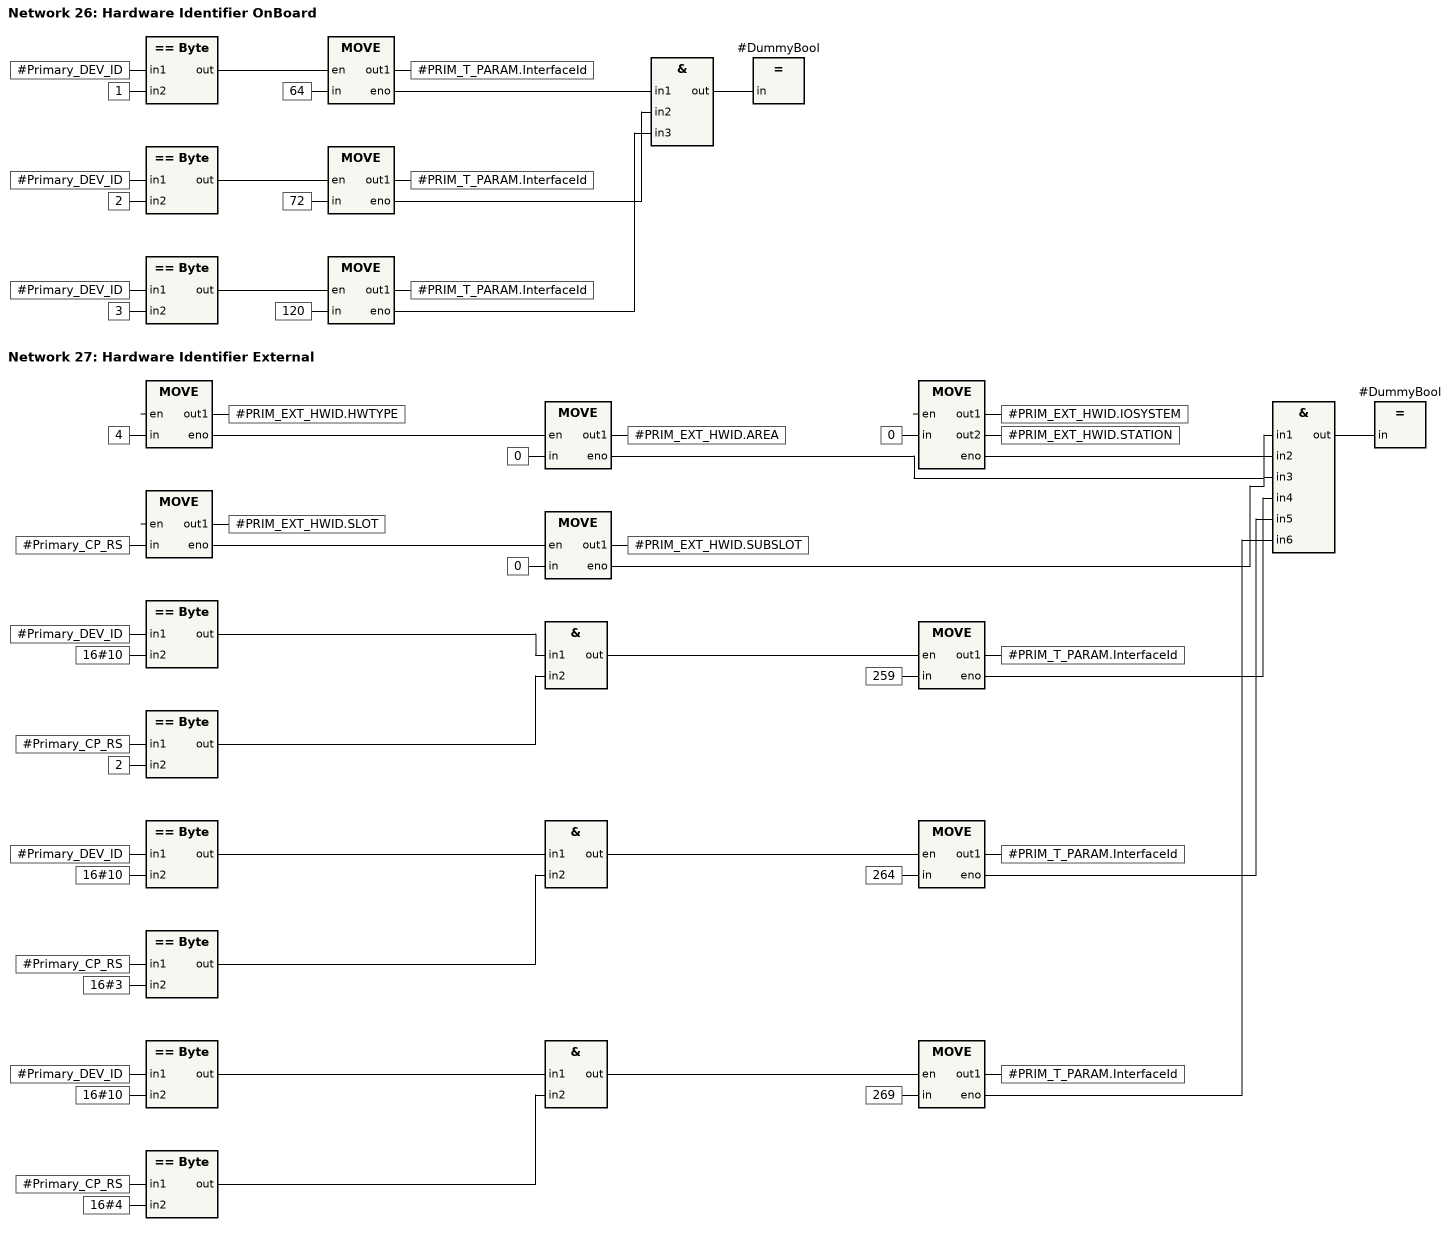
   #_w1 := #Primary_DEV_ID = 1;
   IF #_w1 THEN #PRIM_T_PARAM.InterfaceId := 64; END_IF;
   #_w2 := #Primary_DEV_ID = 2;
   IF #_w2 THEN #PRIM_T_PARAM.InterfaceId := 72; END_IF;
   #_w3 := #Primary_DEV_ID = 3;
   IF #_w3 THEN #PRIM_T_PARAM.InterfaceId := 120; END_IF;
   #DummyBool := #_w1 AND #_w2 AND #_w3;
END_REGION

REGION Network 27: Hardware Identifier External
   #PRIM_EXT_HWID.HWTYPE := 4;
   #PRIM_EXT_HWID.AREA := 0;
   #PRIM_EXT_HWID.IOSYSTEM := 0;
   #PRIM_EXT_HWID.STATION := 0;
   #PRIM_EXT_HWID.SLOT := #Primary_CP_RS;
   #PRIM_EXT_HWID.SUBSLOT := 0;
   #_w1 := (#Primary_DEV_ID = 16#10) AND (#Primary_CP_RS = 2);
   IF #_w1 THEN #PRIM_T_PARAM.InterfaceId := 259; END_IF;
   #_w2 := (#Primary_DEV_ID = 16#10) AND (#Primary_CP_RS = 16#3);
   IF #_w2 THEN #PRIM_T_PARAM.InterfaceId := 264; END_IF;
   #_w3 := (#Primary_DEV_ID = 16#10) AND (#Primary_CP_RS = 16#4);
   IF #_w3 THEN #PRIM_T_PARAM.InterfaceId := 269; END_IF;
   #DummyBool := #_w1 AND #_w2 AND #_w3;
END_REGION

REGION Network 28: Initialise TSAP ID Lengths
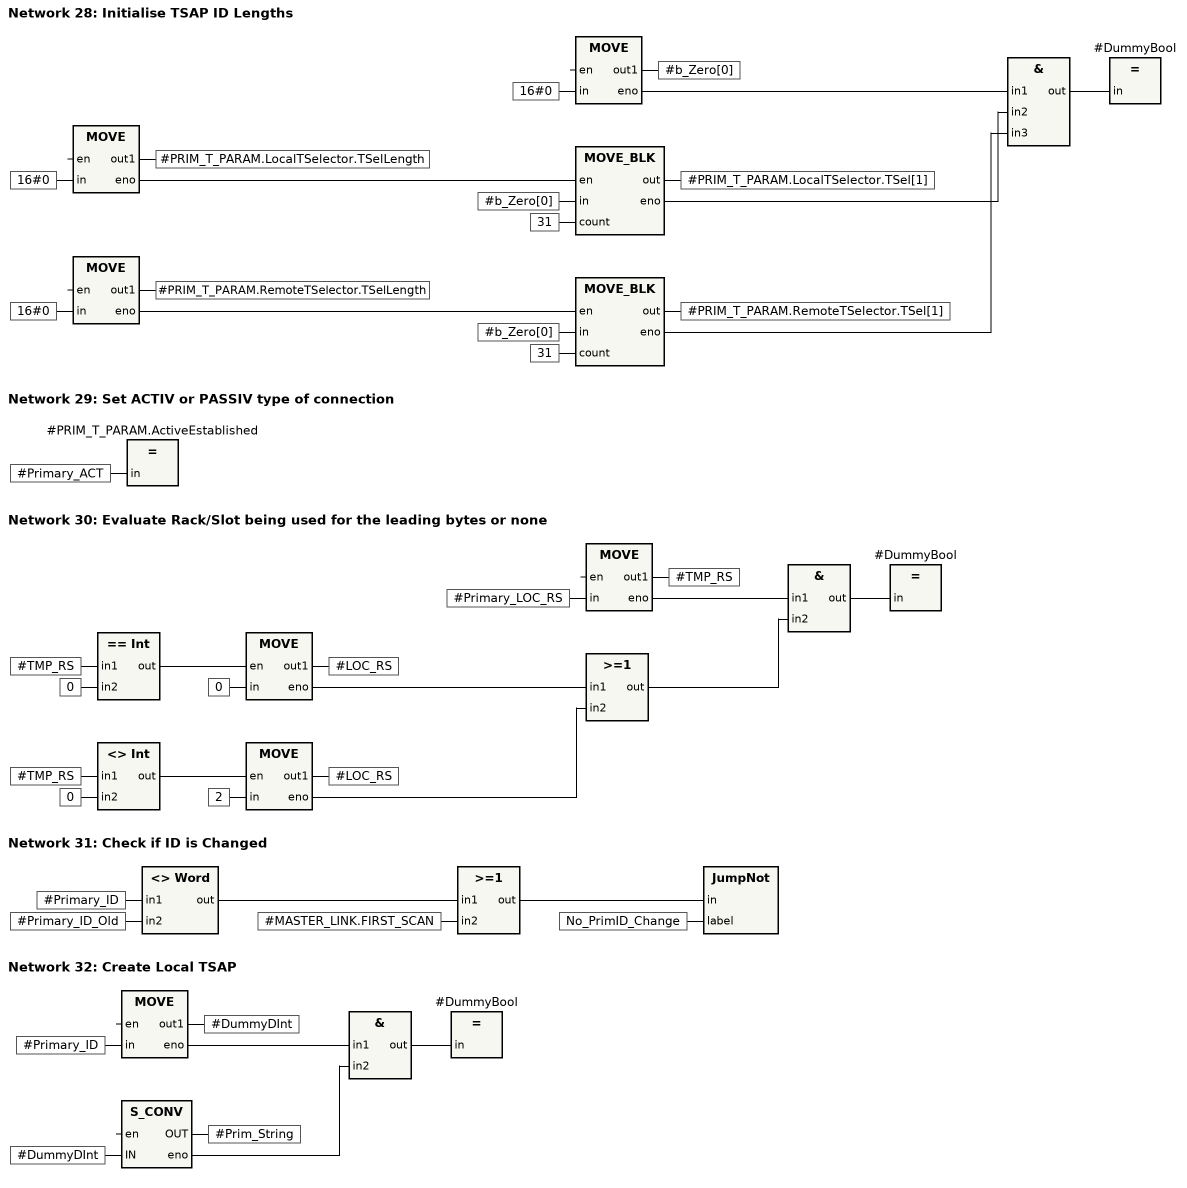
   #b_Zero[0] := 16#0;
   #PRIM_T_PARAM.LocalTSelector.TSelLength := 16#0;
   MOVE_BLK(IN := #b_Zero[0], COUNT := 31, OUT => #PRIM_T_PARAM.LocalTSelector.TSel[1]);
   #PRIM_T_PARAM.RemoteTSelector.TSelLength := 16#0;
   MOVE_BLK(IN := #b_Zero[0], COUNT := 31, OUT => #PRIM_T_PARAM.RemoteTSelector.TSel[1]);
   #DummyBool := TRUE;
END_REGION

REGION Network 29: Set ACTIV or PASSIV type of connection
   // Receive Block Always Pasive
   #PRIM_T_PARAM.ActiveEstablished := #Primary_ACT;
END_REGION

REGION Network 30: Evaluate Rack/Slot being used for the leading bytes or none
   // 1) If R/S = 0 ---> no leading bytes are requested.
   // 2) If R/S # 0 ---> two leading bytes are required.
   // ENO of a box is taken as its EN; it also drops when the box reports an error
   #TMP_RS := #Primary_LOC_RS;
   #_w1 := #TMP_RS = 0;
   IF #_w1 THEN #LOC_RS := 0; END_IF;
   #_w2 := #TMP_RS <> 0;
   IF #_w2 THEN #LOC_RS := 2; END_IF;
   #DummyBool := #_w1 OR #_w2;
END_REGION

REGION Network 31: Check if ID is Changed
   // no SCL statement known for JumpNot: written as a call
   JumpNot(in := (#Primary_ID <> #Primary_ID_Old) OR #MASTER_LINK.FIRST_SCAN, label := No_PrimID_Change);
END_REGION

REGION Network 32: Create Local TSAP
   // Local TSAP = ID_Number
   // ENO of a box is taken as its EN; it also drops when the box reports an error
   #DummyDInt := #Primary_ID;
   #Prim_String := S_CONV(IN := #DummyDInt);
   #DummyBool := TRUE;
END_REGION

REGION Network 33: Check for Empty Space in TSAP
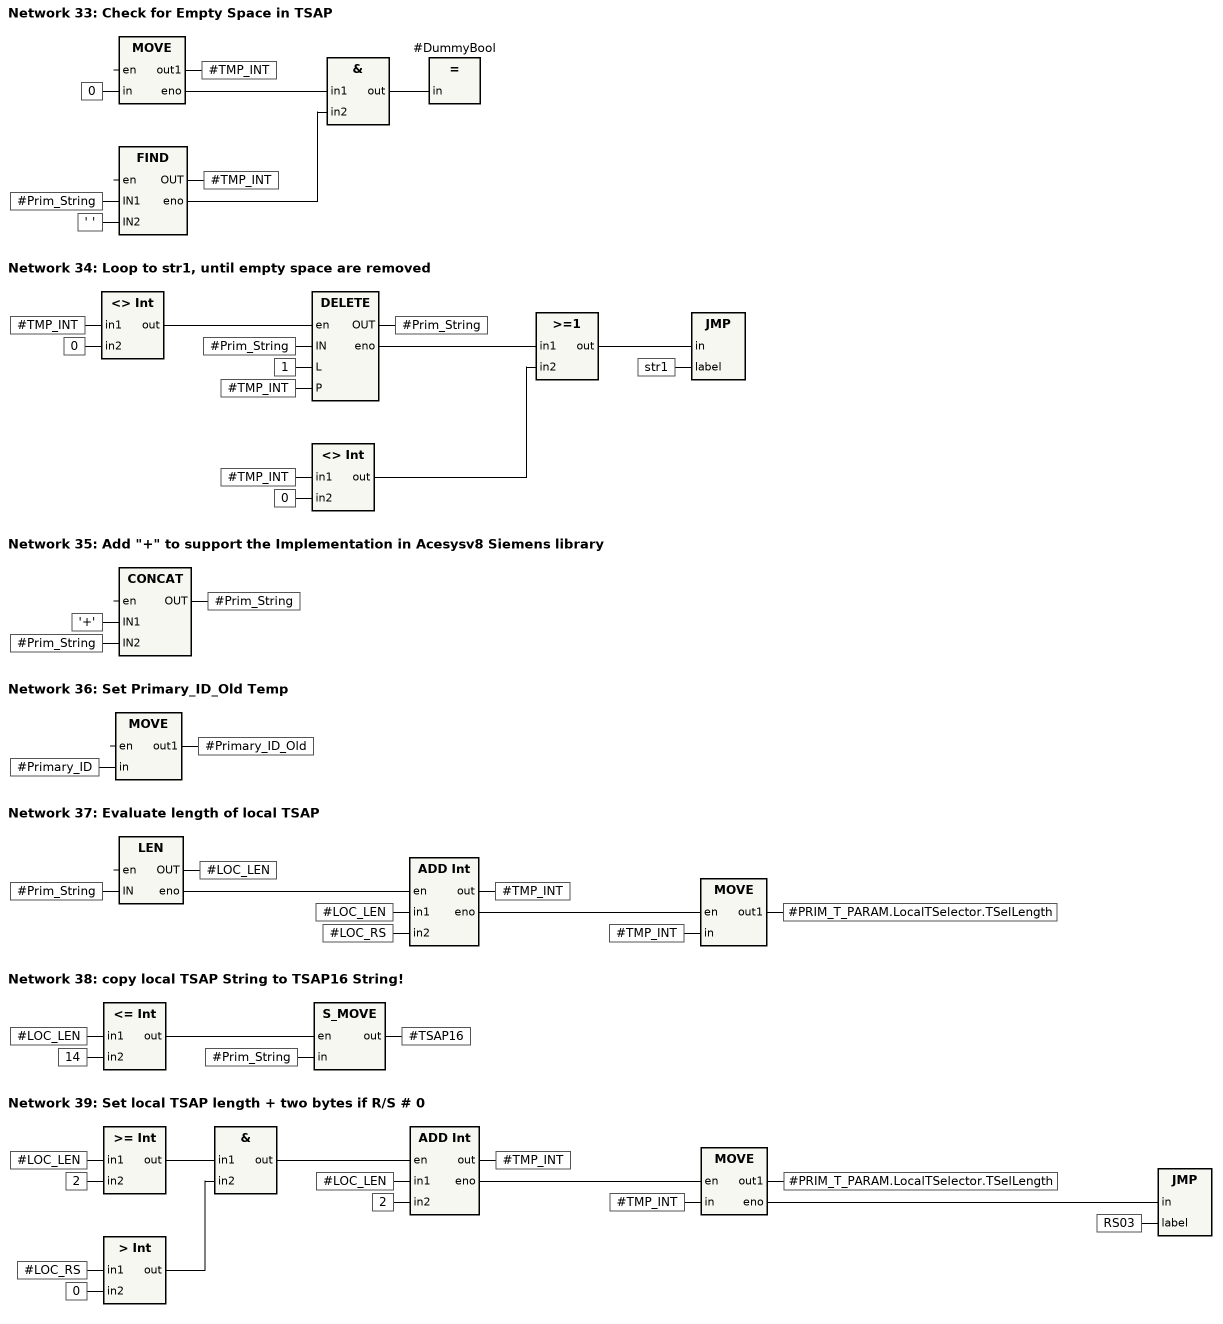
   str1:
   #TMP_INT := 0;
   #TMP_INT := FIND(IN1 := #Prim_String, IN2 := ' ');
   #DummyBool := TRUE;
END_REGION

REGION Network 34: Loop to str1, until empty space are removed
   #_w1 := #TMP_INT <> 0;
   IF #_w1 THEN #Prim_String := DELETE(IN := #Prim_String, L := 1, P := #TMP_INT); END_IF;
   IF #_w1 OR (#TMP_INT <> 0) THEN GOTO str1; END_IF;
END_REGION

REGION Network 35: Add "+" to support the Implementation in Acesysv8 Siemens library
   #Prim_String := CONCAT(IN1 := '+', IN2 := #Prim_String);
END_REGION

REGION Network 36: Set Primary_ID_Old Temp
   No_PrimID_Change:
   #Primary_ID_Old := #Primary_ID;
END_REGION

REGION Network 37: Evaluate length of local TSAP
   // #TSAP.LOC_TSAP
   // ENO of a box is taken as its EN; it also drops when the box reports an error
   #LOC_LEN := LEN(IN := #Prim_String);
   #TMP_INT := #LOC_LEN + #LOC_RS;
   #PRIM_T_PARAM.LocalTSelector.TSelLength := #TMP_INT;
END_REGION

REGION Network 38: copy local TSAP String to TSAP16 String!
   // #TSAP.LOC_TSAP
   IF #LOC_LEN <= 14 THEN #TSAP16 := #Prim_String; END_IF;
END_REGION

REGION Network 39: Set local TSAP length + two bytes if R/S # 0
   #_w1 := (#LOC_LEN >= 2) AND (#LOC_RS > 0);
   IF #_w1 THEN
       #TMP_INT := #LOC_LEN + 2;
       #PRIM_T_PARAM.LocalTSelector.TSelLength := #TMP_INT;
       GOTO RS03;
   END_IF;
END_REGION

REGION Network 40: Set local TSAP values [1 .. 16]
   // Fill in the entire local TSAP (without leading bytes)
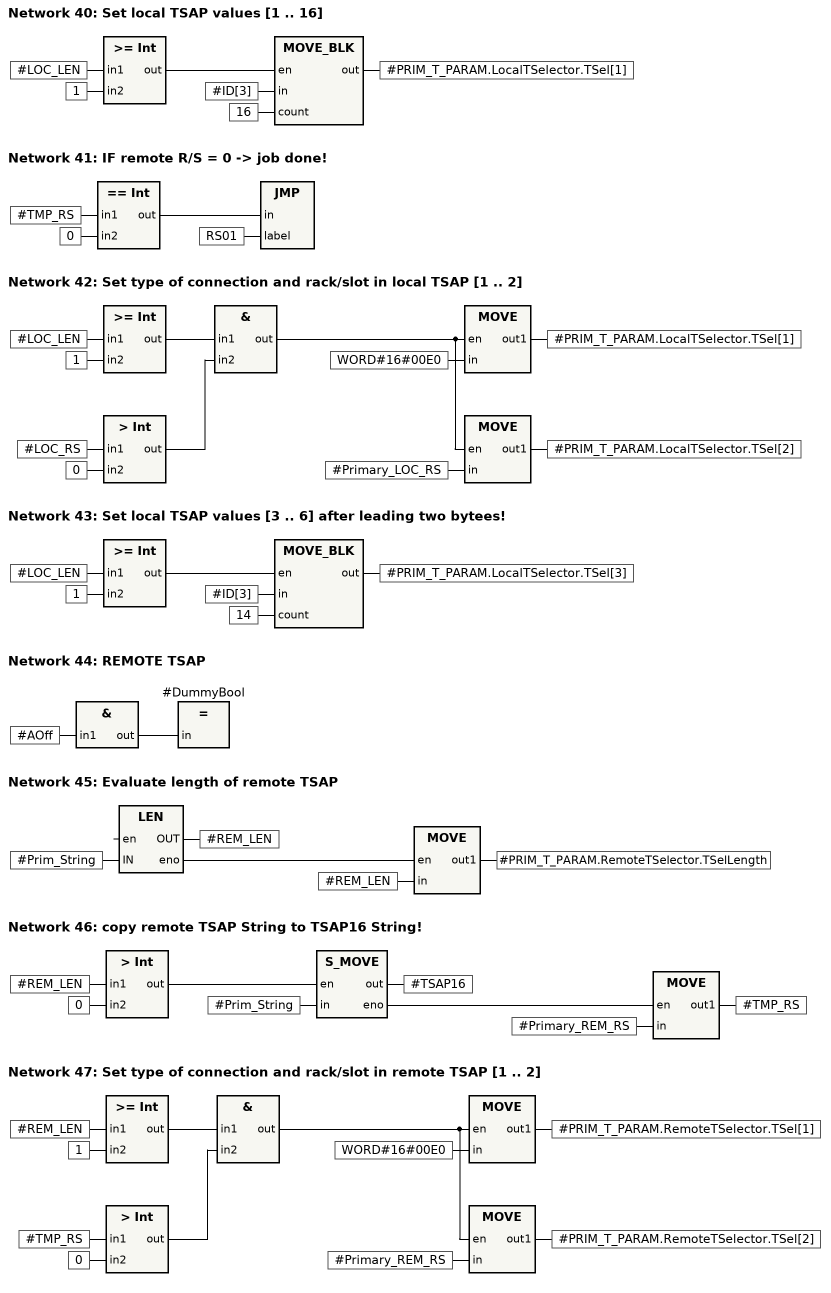
   IF #LOC_LEN >= 1 THEN
       MOVE_BLK(IN := #ID[3], COUNT := 16, OUT => #PRIM_T_PARAM.LocalTSelector.TSel[1]);
   END_IF;
END_REGION

REGION Network 41: IF remote R/S = 0 -> job done!
   IF #TMP_RS = 0 THEN GOTO RS01; END_IF;
END_REGION

REGION Network 42: Set type of connection and rack/slot in local TSAP [1 .. 2]
   // B#16#E0 -> type of connection 
   // B#16#02 -> rack/slot of CPU
   RS03:
   IF (#LOC_LEN >= 1) AND (#LOC_RS > 0) THEN
       #PRIM_T_PARAM.LocalTSelector.TSel[1] := WORD#16#00E0;
       #PRIM_T_PARAM.LocalTSelector.TSel[2] := #Primary_LOC_RS;
   END_IF;
END_REGION

REGION Network 43: Set local TSAP values [3 .. 6] after leading two bytees!
   IF #LOC_LEN >= 1 THEN
       MOVE_BLK(IN := #ID[3], COUNT := 14, OUT => #PRIM_T_PARAM.LocalTSelector.TSel[3]);
   END_IF;
END_REGION

REGION Network 44: REMOTE TSAP
   RS01:
   #DummyBool := #AOff;
END_REGION

REGION Network 45: Evaluate length of remote TSAP
   // Remote TSAP = Local TSAP (DummyString1)
   #REM_LEN := LEN(IN := #Prim_String);
   #PRIM_T_PARAM.RemoteTSelector.TSelLength := #REM_LEN;
END_REGION

REGION Network 46: copy remote TSAP String to TSAP16 String!
   // Remote TSAP = Local TSAP (DummyString1)
   IF #REM_LEN > 0 THEN
       #TSAP16 := #Prim_String;
       #TMP_RS := #Primary_REM_RS;
   END_IF;
END_REGION

REGION Network 47: Set type of connection and rack/slot in remote TSAP [1 .. 2]
   // B#16#E0 -> type of connection, B#16#02 -> rack/slot of CPU
   IF (#REM_LEN >= 1) AND (#TMP_RS > 0) THEN
       #PRIM_T_PARAM.RemoteTSelector.TSel[1] := WORD#16#00E0;
       #PRIM_T_PARAM.RemoteTSelector.TSel[2] := #Primary_REM_RS;
   END_IF;
END_REGION

REGION Network 48: Set remote TSAP length
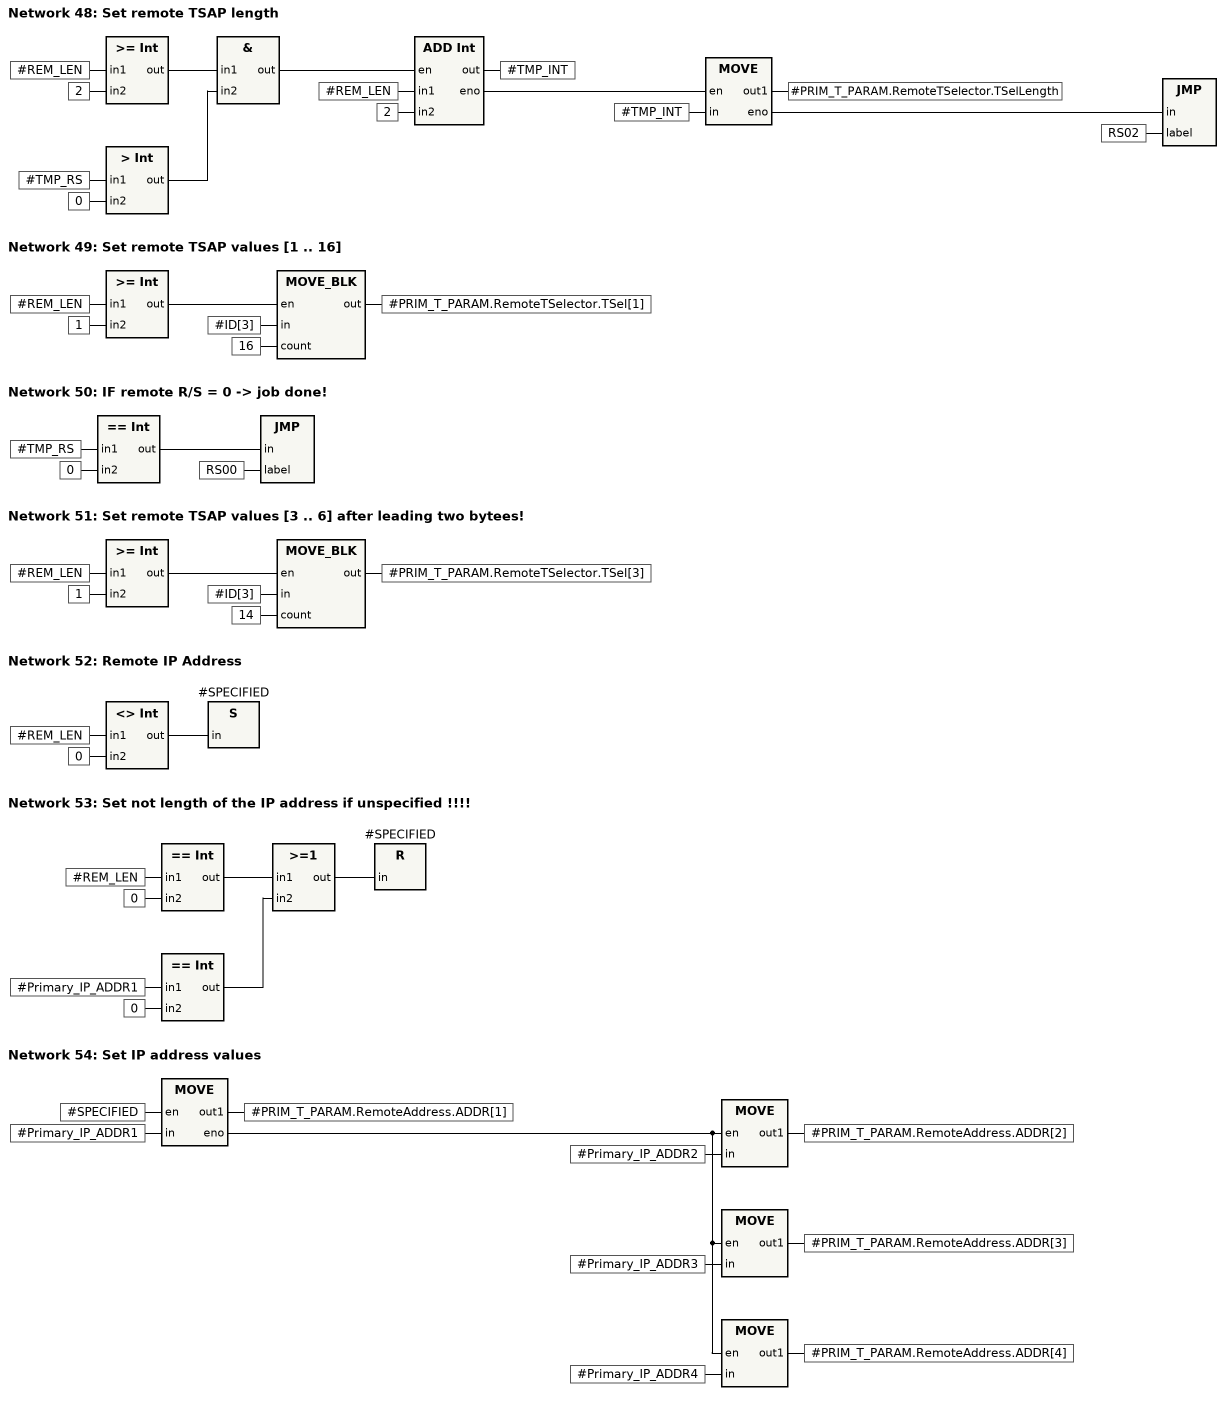
   #_w1 := (#REM_LEN >= 2) AND (#TMP_RS > 0);
   IF #_w1 THEN
       #TMP_INT := #REM_LEN + 2;
       #PRIM_T_PARAM.RemoteTSelector.TSelLength := #TMP_INT;
       GOTO RS02;
   END_IF;
END_REGION

REGION Network 49: Set remote TSAP values [1 .. 16]
   // Fill in the entire local TSAP (without leading bytes)
   IF #REM_LEN >= 1 THEN
       MOVE_BLK(IN := #ID[3], COUNT := 16, OUT => #PRIM_T_PARAM.RemoteTSelector.TSel[1]);
   END_IF;
END_REGION

REGION Network 50: IF remote R/S = 0 -> job done!
   IF #TMP_RS = 0 THEN GOTO RS00; END_IF;
END_REGION

REGION Network 51: Set remote TSAP values [3 .. 6] after leading two bytees!
   RS02:
   IF #REM_LEN >= 1 THEN
       MOVE_BLK(IN := #ID[3], COUNT := 14, OUT => #PRIM_T_PARAM.RemoteTSelector.TSel[3]);
   END_IF;
END_REGION

REGION Network 52: Remote IP Address
   // Set length of the IP address if full-specified only !
   RS00:
   IF #REM_LEN <> 0 THEN #SPECIFIED := TRUE; END_IF;
END_REGION

REGION Network 53: Set not length of the IP address if unspecified !!!!
   // The remote IP address must be zero if
   // 1) remote TSAP is unspecified, or
   // 2) IP address is set up with zero!
   IF (#REM_LEN = 0) OR (#Primary_IP_ADDR1 = 0) THEN #SPECIFIED := FALSE; END_IF;
END_REGION

REGION Network 54: Set IP address values
   // ENO of a box is taken as its EN; it also drops when the box reports an error
   IF #SPECIFIED THEN
       #PRIM_T_PARAM.RemoteAddress.ADDR[1] := #Primary_IP_ADDR1;
       #PRIM_T_PARAM.RemoteAddress.ADDR[2] := #Primary_IP_ADDR2;
       #PRIM_T_PARAM.RemoteAddress.ADDR[3] := #Primary_IP_ADDR3;
       #PRIM_T_PARAM.RemoteAddress.ADDR[4] := #Primary_IP_ADDR4;
   END_IF;
END_REGION

REGION Network 55: <<<<<<<<<<SECONDARY>>>>>>>>>>
END_REGION

REGION Network 56: Hardware Identifier OnBoard
   // Build 002 viv-in 15 Feb 2022 -  X2 Port number corrected.
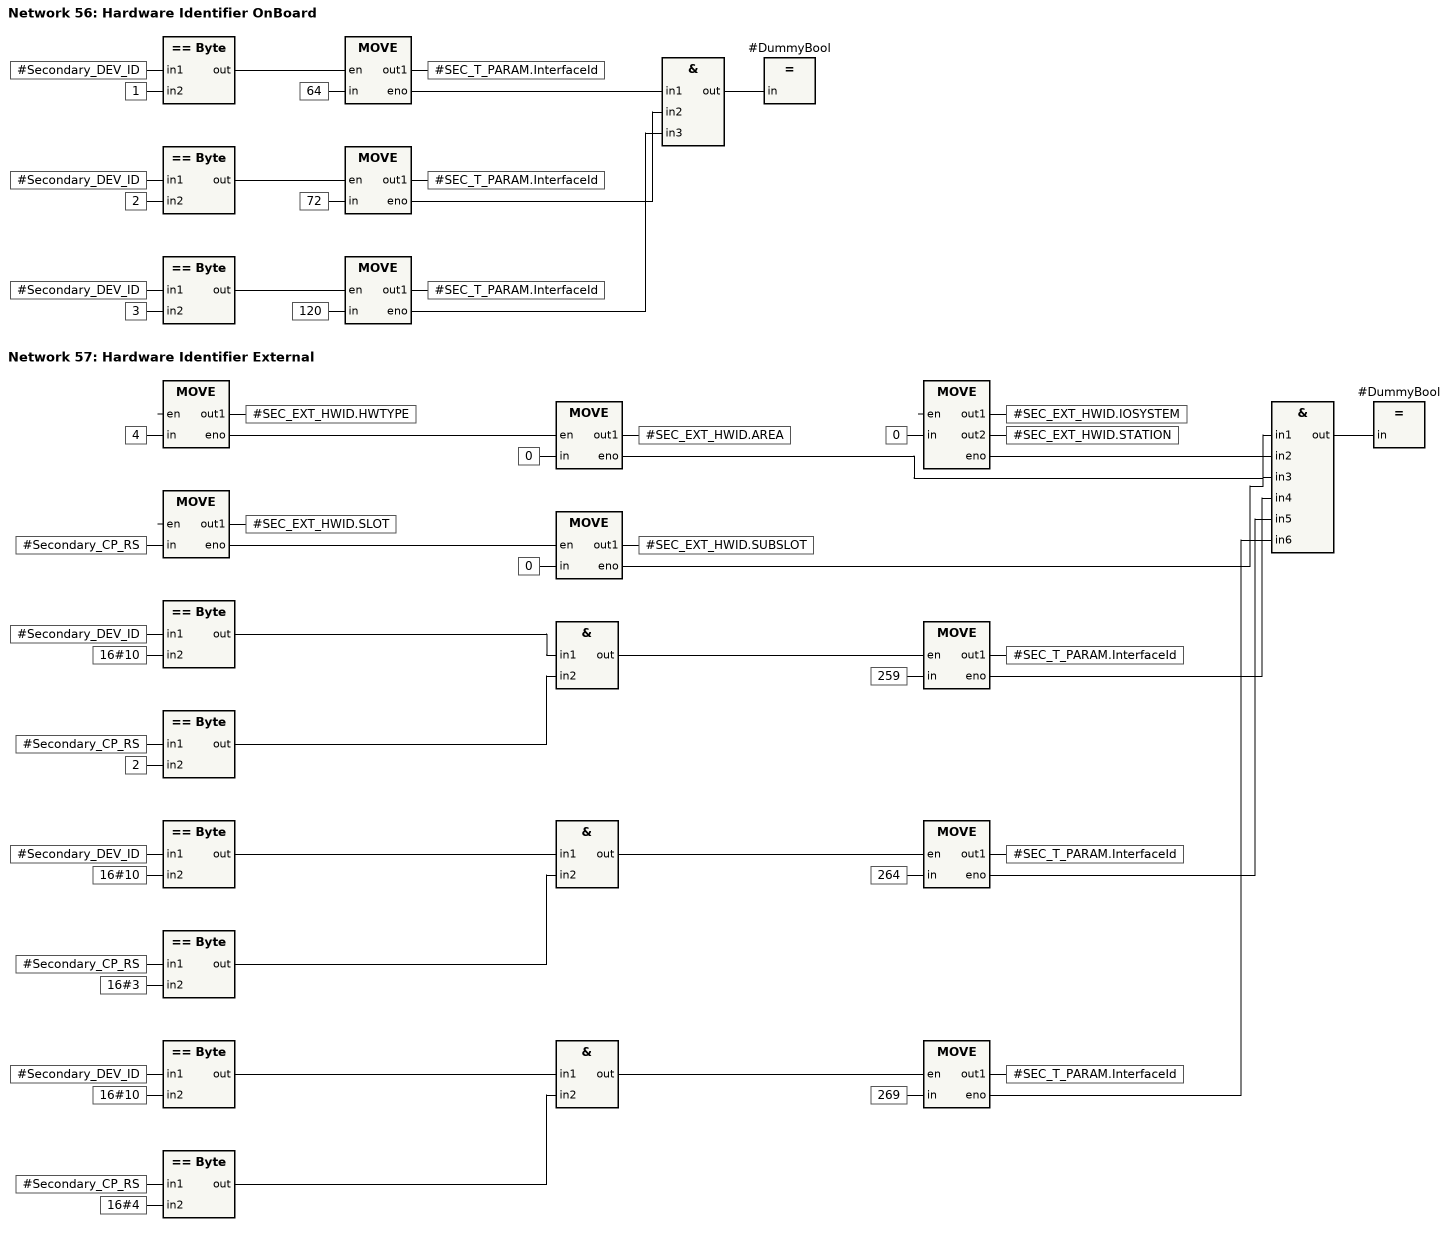
   #_w1 := #Secondary_DEV_ID = 1;
   IF #_w1 THEN #SEC_T_PARAM.InterfaceId := 64; END_IF;
   #_w2 := #Secondary_DEV_ID = 2;
   IF #_w2 THEN #SEC_T_PARAM.InterfaceId := 72; END_IF;
   #_w3 := #Secondary_DEV_ID = 3;
   IF #_w3 THEN #SEC_T_PARAM.InterfaceId := 120; END_IF;
   #DummyBool := #_w1 AND #_w2 AND #_w3;
END_REGION

REGION Network 57: Hardware Identifier External
   #SEC_EXT_HWID.HWTYPE := 4;
   #SEC_EXT_HWID.AREA := 0;
   #SEC_EXT_HWID.IOSYSTEM := 0;
   #SEC_EXT_HWID.STATION := 0;
   #SEC_EXT_HWID.SLOT := #Secondary_CP_RS;
   #SEC_EXT_HWID.SUBSLOT := 0;
   #_w1 := (#Secondary_DEV_ID = 16#10) AND (#Secondary_CP_RS = 2);
   IF #_w1 THEN #SEC_T_PARAM.InterfaceId := 259; END_IF;
   #_w2 := (#Secondary_DEV_ID = 16#10) AND (#Secondary_CP_RS = 16#3);
   IF #_w2 THEN #SEC_T_PARAM.InterfaceId := 264; END_IF;
   #_w3 := (#Secondary_DEV_ID = 16#10) AND (#Secondary_CP_RS = 16#4);
   IF #_w3 THEN #SEC_T_PARAM.InterfaceId := 269; END_IF;
   #DummyBool := #_w1 AND #_w2 AND #_w3;
END_REGION

REGION Network 58: Initialise TSAP
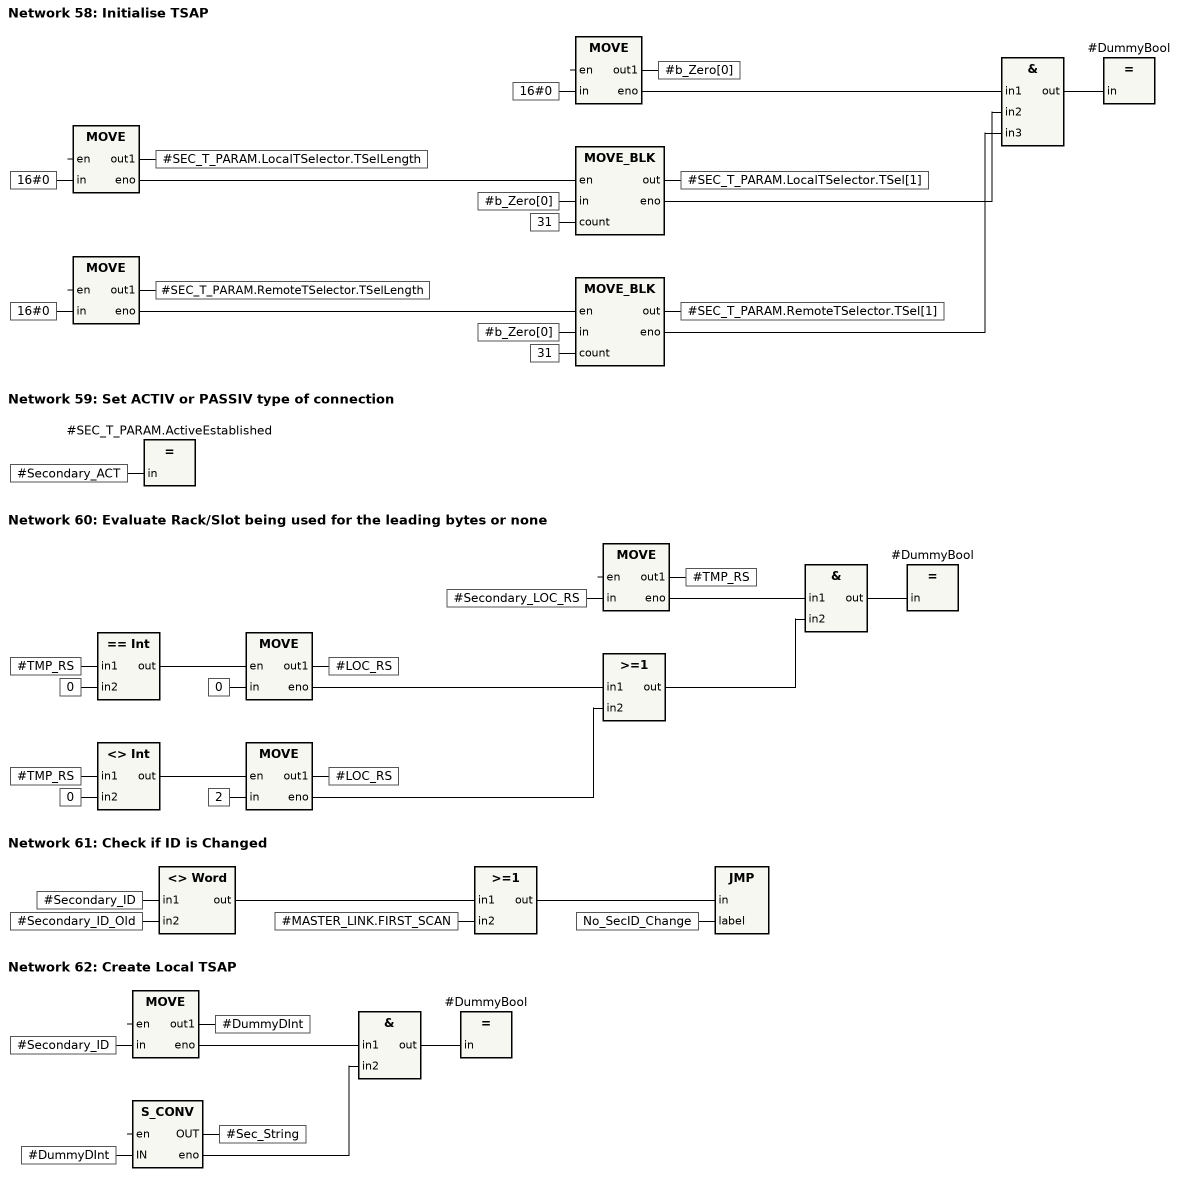
   #b_Zero[0] := 16#0;
   #SEC_T_PARAM.LocalTSelector.TSelLength := 16#0;
   MOVE_BLK(IN := #b_Zero[0], COUNT := 31, OUT => #SEC_T_PARAM.LocalTSelector.TSel[1]);
   #SEC_T_PARAM.RemoteTSelector.TSelLength := 16#0;
   MOVE_BLK(IN := #b_Zero[0], COUNT := 31, OUT => #SEC_T_PARAM.RemoteTSelector.TSel[1]);
   #DummyBool := TRUE;
END_REGION

REGION Network 59: Set ACTIV or PASSIV type of connection
   // Send Block Always Active
   #SEC_T_PARAM.ActiveEstablished := #Secondary_ACT;
END_REGION

REGION Network 60: Evaluate Rack/Slot being used for the leading bytes or none
   // 1) If R/S = 0 ---> no leading bytes are requested.
   // 2) If R/S # 0 ---> two leading bytes are required.
   // ENO of a box is taken as its EN; it also drops when the box reports an error
   #TMP_RS := #Secondary_LOC_RS;
   #_w1 := #TMP_RS = 0;
   IF #_w1 THEN #LOC_RS := 0; END_IF;
   #_w2 := #TMP_RS <> 0;
   IF #_w2 THEN #LOC_RS := 2; END_IF;
   #DummyBool := #_w1 OR #_w2;
END_REGION

REGION Network 61: Check if ID is Changed
   IF (#Secondary_ID <> #Secondary_ID_Old) OR #MASTER_LINK.FIRST_SCAN THEN GOTO No_SecID_Change; END_IF;
END_REGION

REGION Network 62: Create Local TSAP
   // Local TSAP = ID_Number
   // ENO of a box is taken as its EN; it also drops when the box reports an error
   #DummyDInt := #Secondary_ID;
   #Sec_String := S_CONV(IN := #DummyDInt);
   #DummyBool := TRUE;
END_REGION

REGION Network 63: Check for Empty Space in TSAP
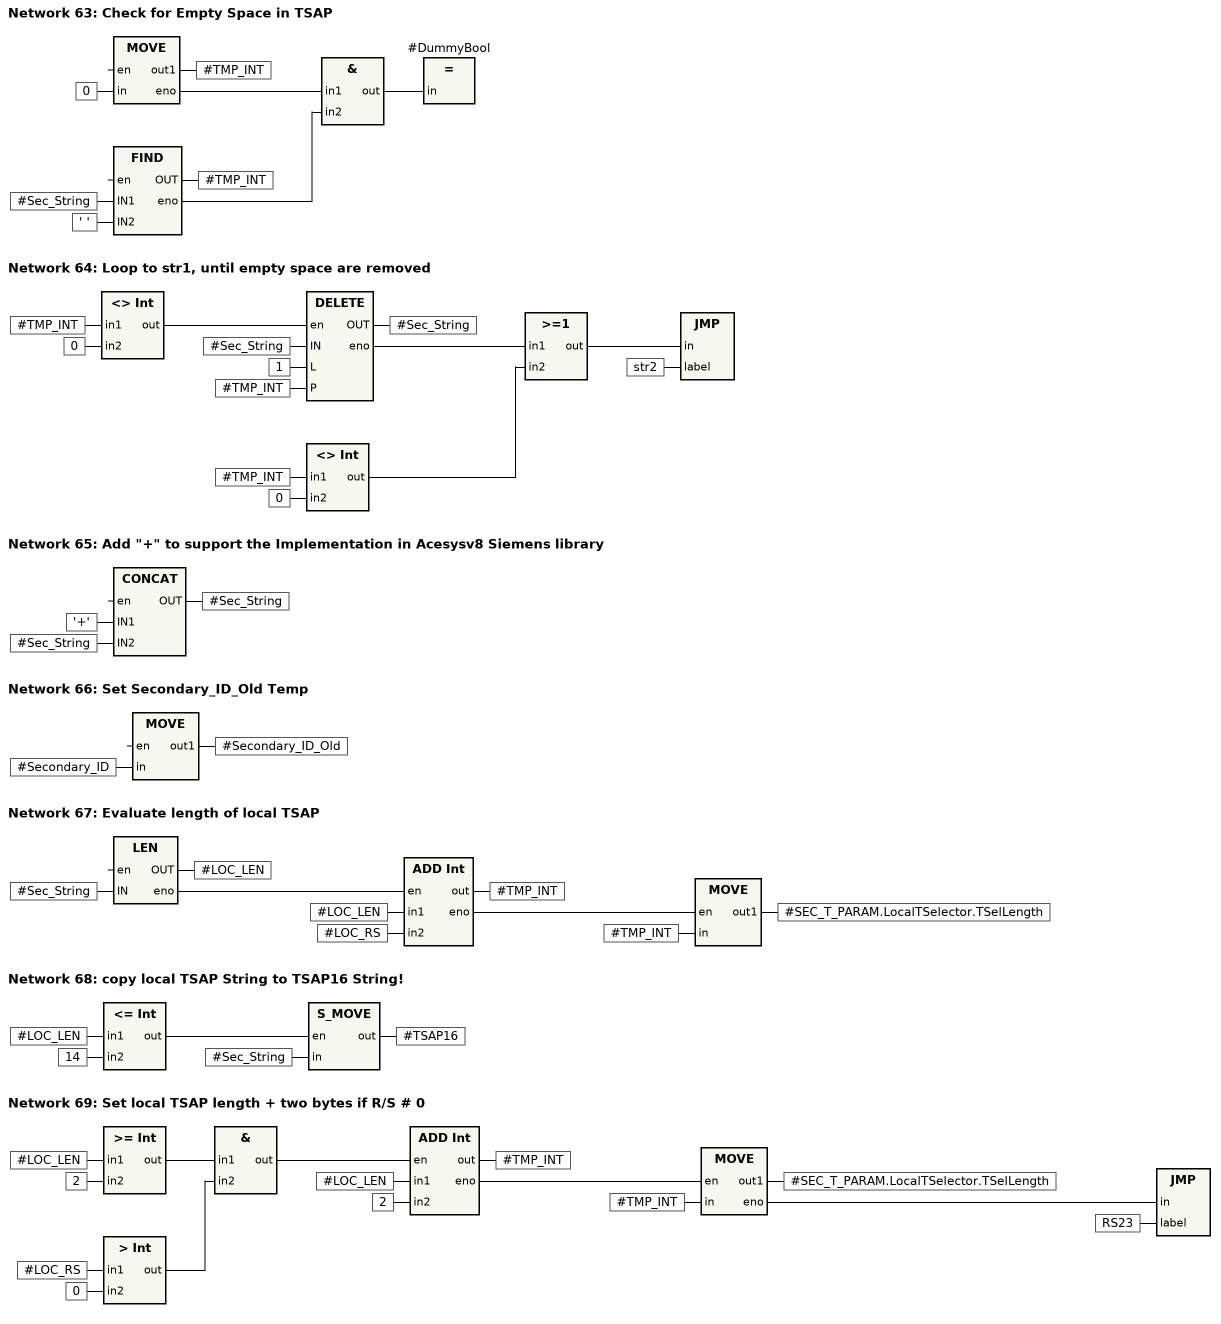
   str2:
   #TMP_INT := 0;
   #TMP_INT := FIND(IN1 := #Sec_String, IN2 := ' ');
   #DummyBool := TRUE;
END_REGION

REGION Network 64: Loop to str1, until empty space are removed
   #_w1 := #TMP_INT <> 0;
   IF #_w1 THEN #Sec_String := DELETE(IN := #Sec_String, L := 1, P := #TMP_INT); END_IF;
   IF #_w1 OR (#TMP_INT <> 0) THEN GOTO str2; END_IF;
END_REGION

REGION Network 65: Add "+" to support the Implementation in Acesysv8 Siemens library
   #Sec_String := CONCAT(IN1 := '+', IN2 := #Sec_String);
END_REGION

REGION Network 66: Set Secondary_ID_Old Temp
   No_SecID_Change:
   #Secondary_ID_Old := #Secondary_ID;
END_REGION

REGION Network 67: Evaluate length of local TSAP
   // #TSAP.LOC_TSAP
   // ENO of a box is taken as its EN; it also drops when the box reports an error
   #LOC_LEN := LEN(IN := #Sec_String);
   #TMP_INT := #LOC_LEN + #LOC_RS;
   #SEC_T_PARAM.LocalTSelector.TSelLength := #TMP_INT;
END_REGION

REGION Network 68: copy local TSAP String to TSAP16 String!
   // #TSAP.LOC_TSAP
   IF #LOC_LEN <= 14 THEN #TSAP16 := #Sec_String; END_IF;
END_REGION

REGION Network 69: Set local TSAP length + two bytes if R/S # 0
   #_w1 := (#LOC_LEN >= 2) AND (#LOC_RS > 0);
   IF #_w1 THEN
       #TMP_INT := #LOC_LEN + 2;
       #SEC_T_PARAM.LocalTSelector.TSelLength := #TMP_INT;
       GOTO RS23;
   END_IF;
END_REGION

REGION Network 70: Set local TSAP values [1 .. 16]
   // Fill in the entire local TSAP (without leading bytes)
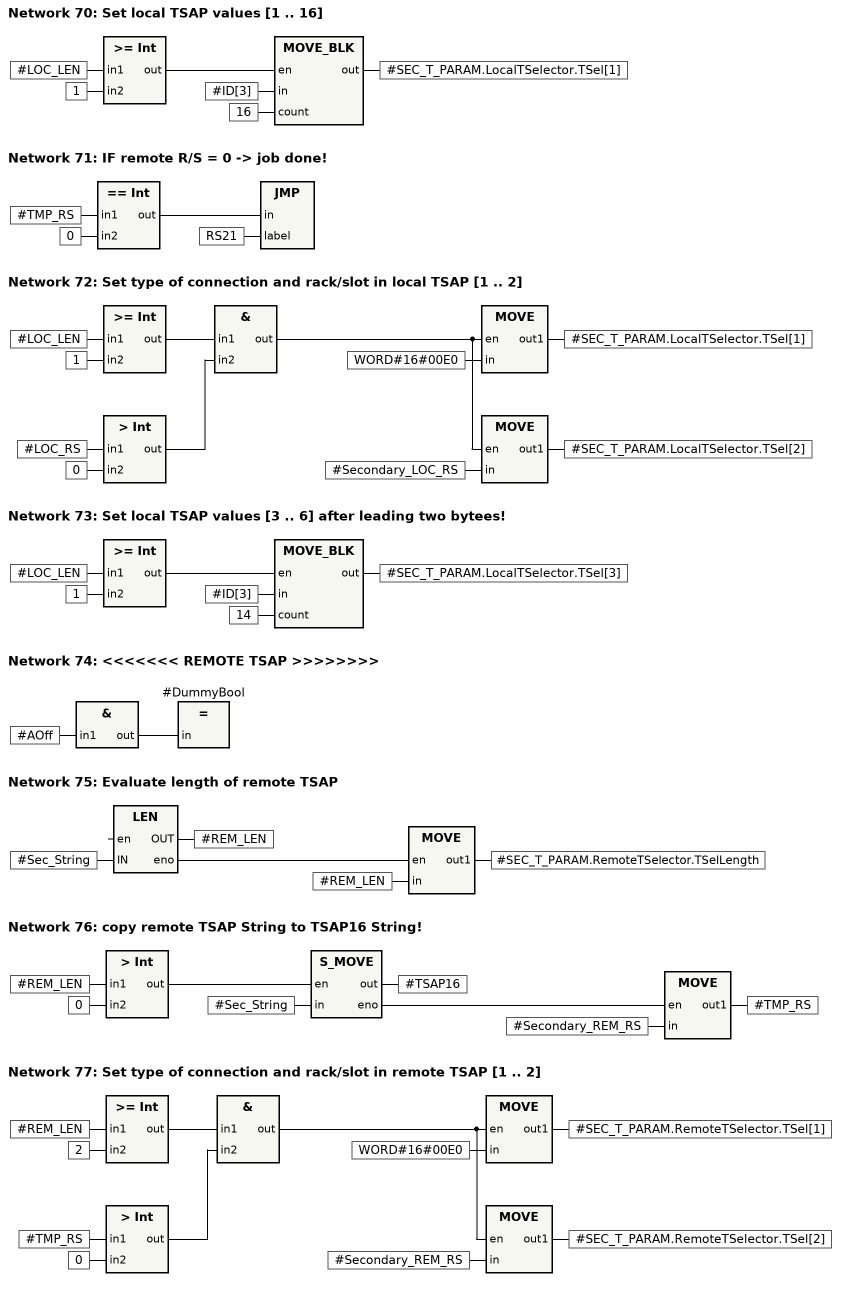
   IF #LOC_LEN >= 1 THEN
       MOVE_BLK(IN := #ID[3], COUNT := 16, OUT => #SEC_T_PARAM.LocalTSelector.TSel[1]);
   END_IF;
END_REGION

REGION Network 71: IF remote R/S = 0 -> job done!
   IF #TMP_RS = 0 THEN GOTO RS21; END_IF;
END_REGION

REGION Network 72: Set type of connection and rack/slot in local TSAP [1 .. 2]
   // B#16#E0 -> type of connection 
   // B#16#02 -> rack/slot of CPU
   RS23:
   IF (#LOC_LEN >= 1) AND (#LOC_RS > 0) THEN
       #SEC_T_PARAM.LocalTSelector.TSel[1] := WORD#16#00E0;
       #SEC_T_PARAM.LocalTSelector.TSel[2] := #Secondary_LOC_RS;
   END_IF;
END_REGION

REGION Network 73: Set local TSAP values [3 .. 6] after leading two bytees!
   IF #LOC_LEN >= 1 THEN
       MOVE_BLK(IN := #ID[3], COUNT := 14, OUT => #SEC_T_PARAM.LocalTSelector.TSel[3]);
   END_IF;
END_REGION

REGION Network 74: <<<<<<< REMOTE TSAP >>>>>>>>
   RS21:
   #DummyBool := #AOff;
END_REGION

REGION Network 75: Evaluate length of remote TSAP
   // Remote TSAP = Local TSAP (DummyString1)
   #REM_LEN := LEN(IN := #Sec_String);
   #SEC_T_PARAM.RemoteTSelector.TSelLength := #REM_LEN;
END_REGION

REGION Network 76: copy remote TSAP String to TSAP16 String!
   // Remote TSAP = Local TSAP (DummyString)
   IF #REM_LEN > 0 THEN
       #TSAP16 := #Sec_String;
       #TMP_RS := #Secondary_REM_RS;
   END_IF;
END_REGION

REGION Network 77: Set type of connection and rack/slot in remote TSAP [1 .. 2]
   // B#16#E0 -> type of connection 
   // B#16#02 -> rack/slot of CPU
   IF (#REM_LEN >= 2) AND (#TMP_RS > 0) THEN
       #SEC_T_PARAM.RemoteTSelector.TSel[1] := WORD#16#00E0;
       #SEC_T_PARAM.RemoteTSelector.TSel[2] := #Secondary_REM_RS;
   END_IF;
END_REGION

REGION Network 78: Set remote TSAP length
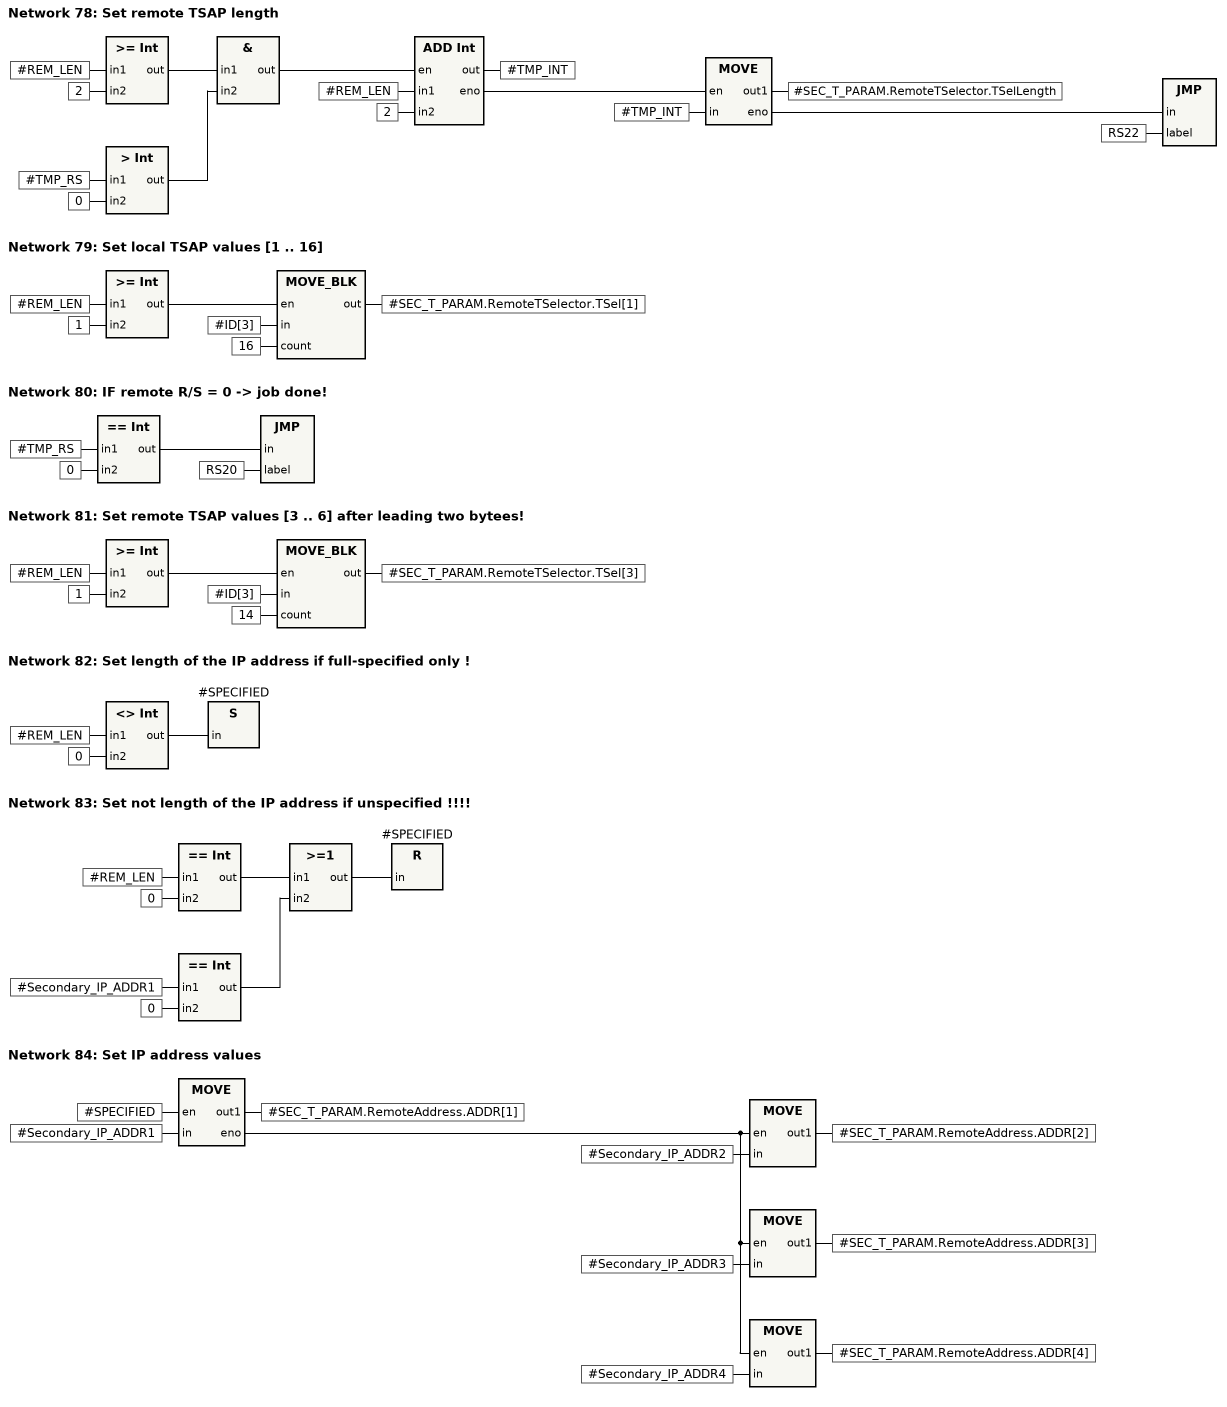
   #_w1 := (#REM_LEN >= 2) AND (#TMP_RS > 0);
   IF #_w1 THEN
       #TMP_INT := #REM_LEN + 2;
       #SEC_T_PARAM.RemoteTSelector.TSelLength := #TMP_INT;
       GOTO RS22;
   END_IF;
END_REGION

REGION Network 79: Set local TSAP values [1 .. 16]
   // Fill in the entire local TSAP (without leading bytes)
   IF #REM_LEN >= 1 THEN
       MOVE_BLK(IN := #ID[3], COUNT := 16, OUT => #SEC_T_PARAM.RemoteTSelector.TSel[1]);
   END_IF;
END_REGION

REGION Network 80: IF remote R/S = 0 -> job done!
   IF #TMP_RS = 0 THEN GOTO RS20; END_IF;
END_REGION

REGION Network 81: Set remote TSAP values [3 .. 6] after leading two bytees!
   RS22:
   IF #REM_LEN >= 1 THEN
       MOVE_BLK(IN := #ID[3], COUNT := 14, OUT => #SEC_T_PARAM.RemoteTSelector.TSel[3]);
   END_IF;
END_REGION

REGION Network 82: Set length of the IP address if full-specified only !
   RS20:
   IF #REM_LEN <> 0 THEN #SPECIFIED := TRUE; END_IF;
END_REGION

REGION Network 83: Set not length of the IP address if unspecified !!!!
   // The remote IP address must be zero if
   // 1) remote TSAP is unspecified, or
   // 2) IP address is set up with zero!
   IF (#REM_LEN = 0) OR (#Secondary_IP_ADDR1 = 0) THEN #SPECIFIED := FALSE; END_IF;
END_REGION

REGION Network 84: Set IP address values
   // ENO of a box is taken as its EN; it also drops when the box reports an error
   IF #SPECIFIED THEN
       #SEC_T_PARAM.RemoteAddress.ADDR[1] := #Secondary_IP_ADDR1;
       #SEC_T_PARAM.RemoteAddress.ADDR[2] := #Secondary_IP_ADDR2;
       #SEC_T_PARAM.RemoteAddress.ADDR[3] := #Secondary_IP_ADDR3;
       #SEC_T_PARAM.RemoteAddress.ADDR[4] := #Secondary_IP_ADDR4;
   END_IF;
END_REGION

REGION Network 85: Establish or register ISO-on_TCP connection
   // After the connection has been established, it is automatically monitored and 
   // maintained by the operating system of the CPU.
   // 
   // If the connection has been interrupted, by any line break or due to the remote 
   // communications partner, the active partner attempts to reestablish the 
   // connection.
   // 
   // Therefore, the FB 65 "TCON" may not be called again!
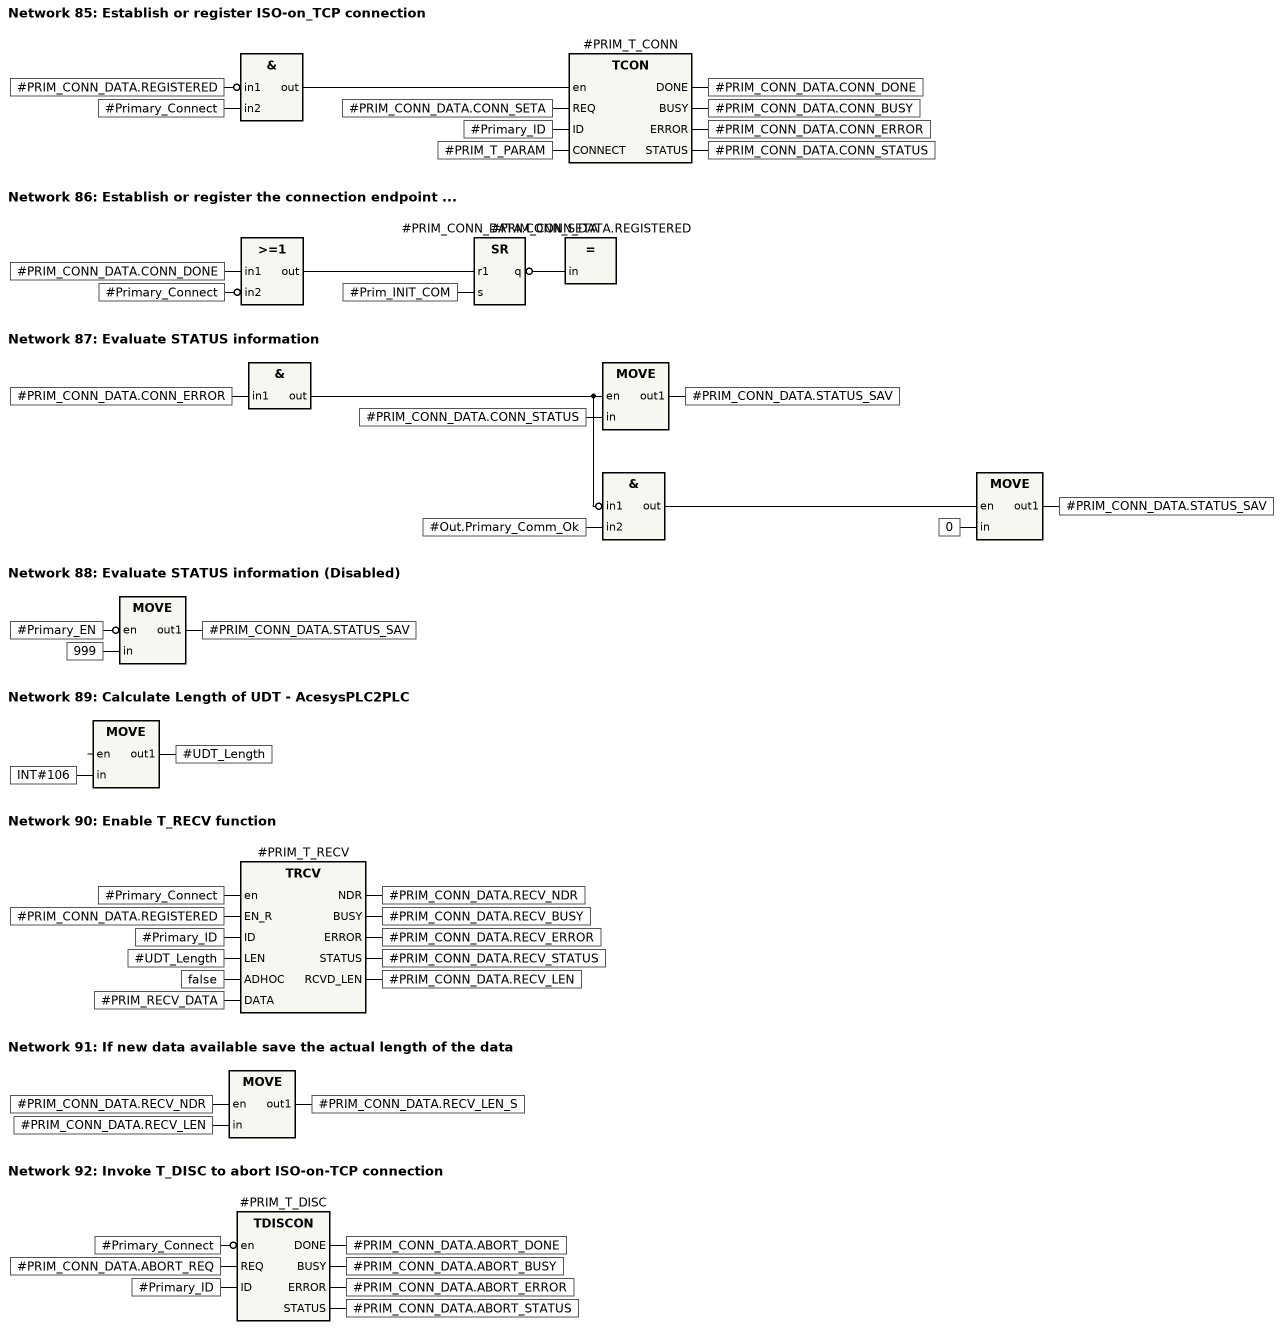
   IF NOT #PRIM_CONN_DATA.REGISTERED AND #Primary_Connect THEN
       #PRIM_T_CONN(REQ := #PRIM_CONN_DATA.CONN_SETA,   // TCON
                    ID := #Primary_ID,
                    CONNECT := #PRIM_T_PARAM,
                    DONE => #PRIM_CONN_DATA.CONN_DONE,
                    BUSY => #PRIM_CONN_DATA.CONN_BUSY,
                    ERROR => #PRIM_CONN_DATA.CONN_ERROR,
                    STATUS => #PRIM_CONN_DATA.CONN_STATUS);
   END_IF;
END_REGION

REGION Network 86: Establish or register the connection endpoint ...
   // while startup phase (initial).
   // 
   // Indication of the connection status:
   // 
   // a) If the CPU may establish the specified connection after Stop/Run  
   // immediately, the variable "REGISTERED" indicates HIGH (=1).
   // 
   // b) If the CPU is not able to establish the specified connection after Stop/Run, 
   // the variable "REGISTERED" remains LOW(=0).
   // 
   // c) Note: If the instance DB is loaded by the user, the variable "REGISTERED" 
   // indicates HIGH, although the connection may not be established yet. 
   // However, the FB64 "TRCV" would indicate the STATUS=0x80C4, as long as the 
   // connection has not been established.
   IF #Prim_INIT_COM THEN
       #PRIM_CONN_DATA.CONN_SETA := TRUE;   // SR flip-flop
   END_IF;
   IF #PRIM_CONN_DATA.CONN_DONE OR NOT #Primary_Connect THEN #PRIM_CONN_DATA.CONN_SETA := FALSE; END_IF;
   #PRIM_CONN_DATA.REGISTERED := NOT #PRIM_CONN_DATA.CONN_SETA;
END_REGION

REGION Network 87: Evaluate STATUS information
   IF #PRIM_CONN_DATA.CONN_ERROR THEN #PRIM_CONN_DATA.STATUS_SAV := #PRIM_CONN_DATA.CONN_STATUS; END_IF;
   IF NOT #PRIM_CONN_DATA.CONN_ERROR AND #Out.Primary_Comm_Ok THEN #PRIM_CONN_DATA.STATUS_SAV := 0; END_IF;
END_REGION

REGION Network 88: Evaluate STATUS information (Disabled)
   IF NOT #Primary_EN THEN #PRIM_CONN_DATA.STATUS_SAV := 999; END_IF;
END_REGION

REGION Network 89: Calculate Length of UDT - AcesysPLC2PLC
   #UDT_Length := INT#106;
END_REGION

REGION Network 90: Enable T_RECV function
   // The data is stored into the buffer specified with the ANY pointer of the 
   // receive buffer (i.e., DATA parameter). After the data has been received, the 
   // data is immediately available in the receive buffer. Receiving is indicated by 
   // the NDR output parameter.
   IF #Primary_Connect THEN
       #PRIM_T_RECV(EN_R := #PRIM_CONN_DATA.REGISTERED,   // TRCV
                    ID := #Primary_ID,
                    LEN := #UDT_Length,
                    ADHOC := false,
                    DATA := #PRIM_RECV_DATA,
                    NDR => #PRIM_CONN_DATA.RECV_NDR,
                    BUSY => #PRIM_CONN_DATA.RECV_BUSY,
                    ERROR => #PRIM_CONN_DATA.RECV_ERROR,
                    STATUS => #PRIM_CONN_DATA.RECV_STATUS,
                    RCVD_LEN => #PRIM_CONN_DATA.RECV_LEN);
   END_IF;
END_REGION

REGION Network 91: If new data available save the actual length of the data
   IF #PRIM_CONN_DATA.RECV_NDR THEN #PRIM_CONN_DATA.RECV_LEN_S := #PRIM_CONN_DATA.RECV_LEN; END_IF;
END_REGION

REGION Network 92: Invoke T_DISC to abort ISO-on-TCP connection
   // The FB 66 "TDISCON" terminates a communications connection from the CPU to a
   // communications partner.
   // 
   // An existing connection is terminated when FB 66 "TDISCON" is called or when the
   // CPU has gone into STOP mode. To reestablish the connection, the FB 65 "TCON" 
   // has to be invoked again.
   IF NOT #Primary_Connect THEN
       #PRIM_T_DISC(REQ := #PRIM_CONN_DATA.ABORT_REQ,   // TDISCON
                    ID := #Primary_ID,
                    DONE => #PRIM_CONN_DATA.ABORT_DONE,
                    BUSY => #PRIM_CONN_DATA.ABORT_BUSY,
                    ERROR => #PRIM_CONN_DATA.ABORT_ERROR,
                    STATUS => #PRIM_CONN_DATA.ABORT_STATUS);
   END_IF;
END_REGION

REGION Network 93: If "ABORT" is set, the connection will be aborted
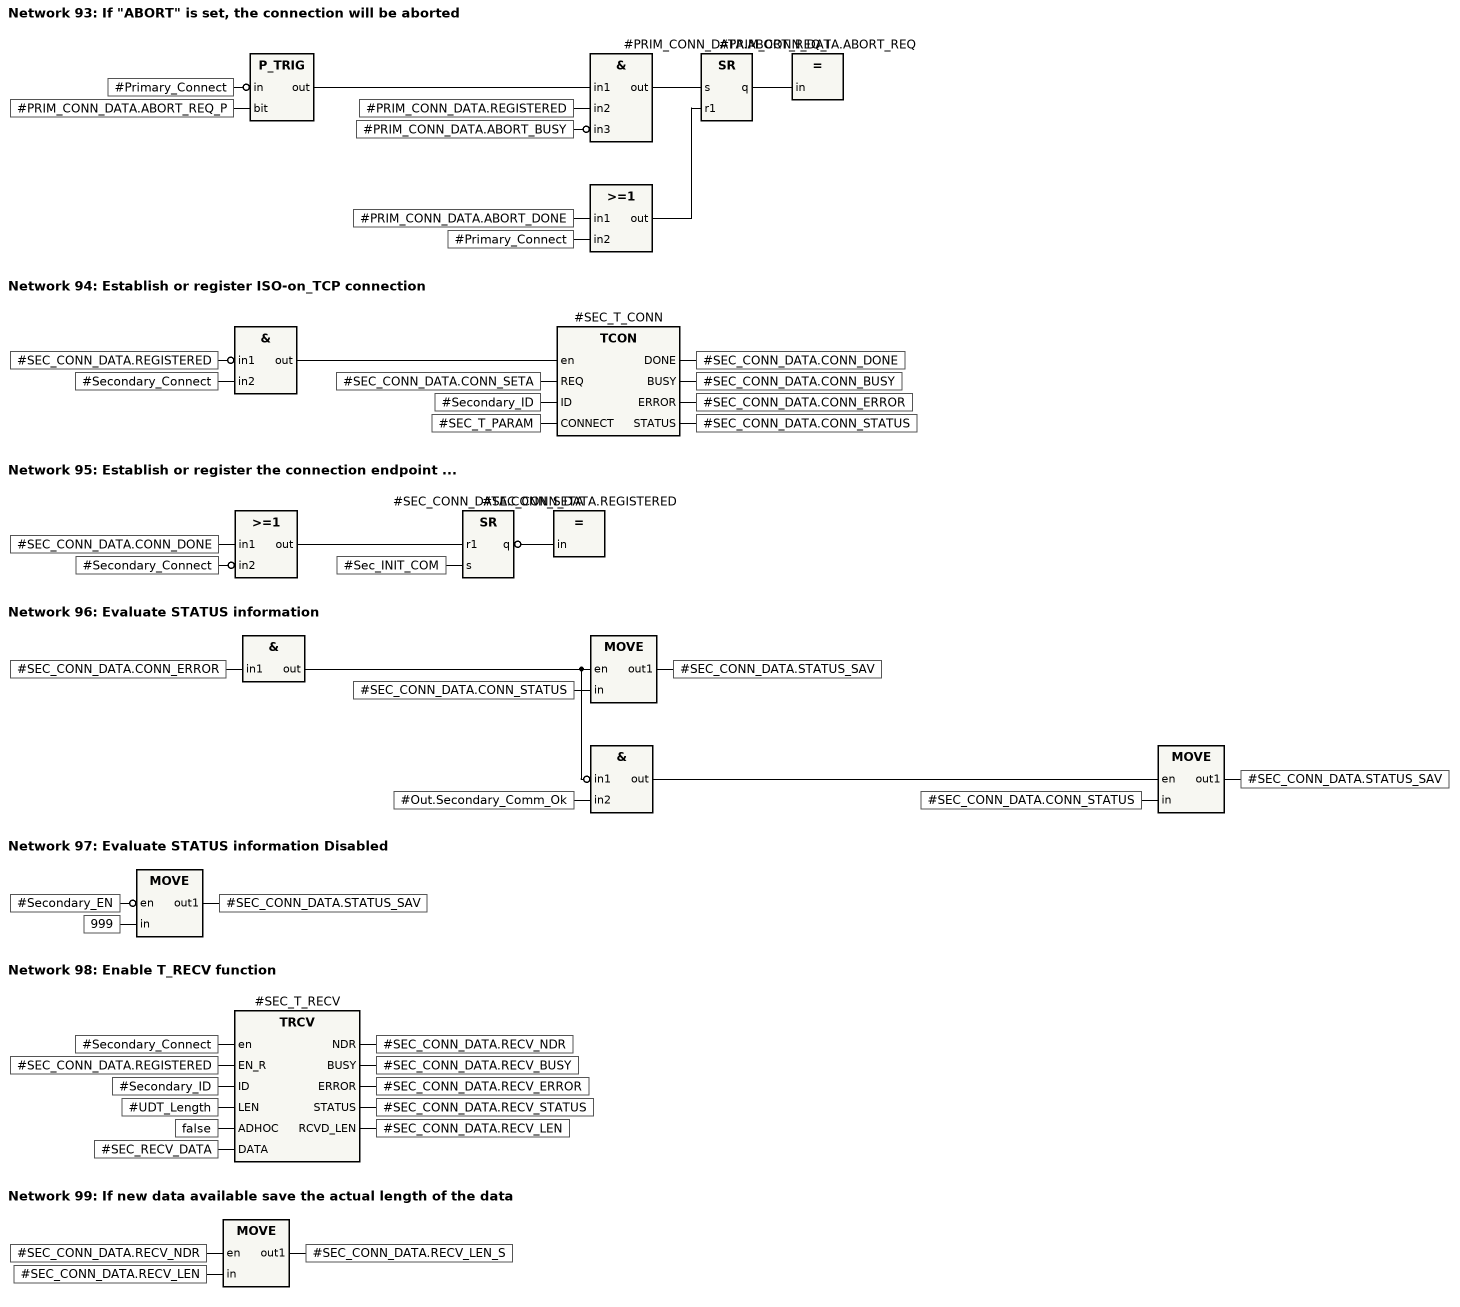
   #_w1 := NOT #Primary_Connect AND NOT #PRIM_CONN_DATA.ABORT_REQ_P;   // rising edge
   #PRIM_CONN_DATA.ABORT_REQ_P := NOT #Primary_Connect;
   IF #_w1 AND #PRIM_CONN_DATA.REGISTERED AND NOT #PRIM_CONN_DATA.ABORT_BUSY THEN
       #PRIM_CONN_DATA.ABORT_REQ_I := TRUE;   // SR flip-flop
   END_IF;
   IF #PRIM_CONN_DATA.ABORT_DONE OR #Primary_Connect THEN #PRIM_CONN_DATA.ABORT_REQ_I := FALSE; END_IF;
   #PRIM_CONN_DATA.ABORT_REQ := #PRIM_CONN_DATA.ABORT_REQ_I;
END_REGION

REGION Network 94: Establish or register ISO-on_TCP connection
   // After the connection has been established, it is automatically monitored and 
   // maintained by the operating system of the CPU.
   // 
   // If the connection has been interrupted, by any line break or due to the remote 
   // communications partner, the active partner attempts to reestablish the 
   // connection.
   // 
   // Therefore, the FB 65 "TCON" may not be called again!
   IF NOT #SEC_CONN_DATA.REGISTERED AND #Secondary_Connect THEN
       #SEC_T_CONN(REQ := #SEC_CONN_DATA.CONN_SETA,   // TCON
                   ID := #Secondary_ID,
                   CONNECT := #SEC_T_PARAM,
                   DONE => #SEC_CONN_DATA.CONN_DONE,
                   BUSY => #SEC_CONN_DATA.CONN_BUSY,
                   ERROR => #SEC_CONN_DATA.CONN_ERROR,
                   STATUS => #SEC_CONN_DATA.CONN_STATUS);
   END_IF;
END_REGION

REGION Network 95: Establish or register the connection endpoint ...
   // while startup phase (initial).
   // 
   // Indication of the connection status:
   // 
   // a) If the CPU may establish the specified connection after Stop/Run  
   // immediately, the variable "REGISTERED" indicates HIGH (=1).
   // 
   // b) If the CPU is not able to establish the specified connection after Stop/Run, 
   // the variable "REGISTERED" remains LOW(=0).
   // 
   // c) Note: If the instance DB is loaded by the user, the variable "REGISTERED" 
   // indicates HIGH, although the connection may not be established yet. 
   // However, the FB64 "TRCV" would indicate the STATUS=0x80C4, as long as the 
   // connection has not been established.
   IF #Sec_INIT_COM THEN
       #SEC_CONN_DATA.CONN_SETA := TRUE;   // SR flip-flop
   END_IF;
   IF #SEC_CONN_DATA.CONN_DONE OR NOT #Secondary_Connect THEN #SEC_CONN_DATA.CONN_SETA := FALSE; END_IF;
   #SEC_CONN_DATA.REGISTERED := NOT #SEC_CONN_DATA.CONN_SETA;
END_REGION

REGION Network 96: Evaluate STATUS information
   IF #SEC_CONN_DATA.CONN_ERROR THEN #SEC_CONN_DATA.STATUS_SAV := #SEC_CONN_DATA.CONN_STATUS; END_IF;
   IF NOT #SEC_CONN_DATA.CONN_ERROR AND #Out.Secondary_Comm_Ok THEN
       #SEC_CONN_DATA.STATUS_SAV := #SEC_CONN_DATA.CONN_STATUS;
   END_IF;
END_REGION

REGION Network 97: Evaluate STATUS information Disabled
   IF NOT #Secondary_EN THEN #SEC_CONN_DATA.STATUS_SAV := 999; END_IF;
END_REGION

REGION Network 98: Enable T_RECV function
   // The data is stored into the buffer specified with the ANY pointer of the 
   // receive buffer (i.e., DATA parameter). After the data has been received, the 
   // data is immediately available in the receive buffer. Receiving is indicated by 
   // the NDR output parameter.
   IF #Secondary_Connect THEN
       #SEC_T_RECV(EN_R := #SEC_CONN_DATA.REGISTERED,   // TRCV
                   ID := #Secondary_ID,
                   LEN := #UDT_Length,
                   ADHOC := false,
                   DATA := #SEC_RECV_DATA,
                   NDR => #SEC_CONN_DATA.RECV_NDR,
                   BUSY => #SEC_CONN_DATA.RECV_BUSY,
                   ERROR => #SEC_CONN_DATA.RECV_ERROR,
                   STATUS => #SEC_CONN_DATA.RECV_STATUS,
                   RCVD_LEN => #SEC_CONN_DATA.RECV_LEN);
   END_IF;
END_REGION

REGION Network 99: If new data available save the actual length of the data
   IF #SEC_CONN_DATA.RECV_NDR THEN #SEC_CONN_DATA.RECV_LEN_S := #SEC_CONN_DATA.RECV_LEN; END_IF;
END_REGION

REGION Network 100: Invoke T_DISC to abort ISO-on-TCP connection
   // The FB 66 "TDISCON" terminates a communications connection from the CPU to a
   // communications partner.
   // 
   // An existing connection is terminated when FB 66 "TDISCON" is called or when the
   // CPU has gone into STOP mode. To reestablish the connection, the FB 65 "TCON" 
   // has to be invoked again.
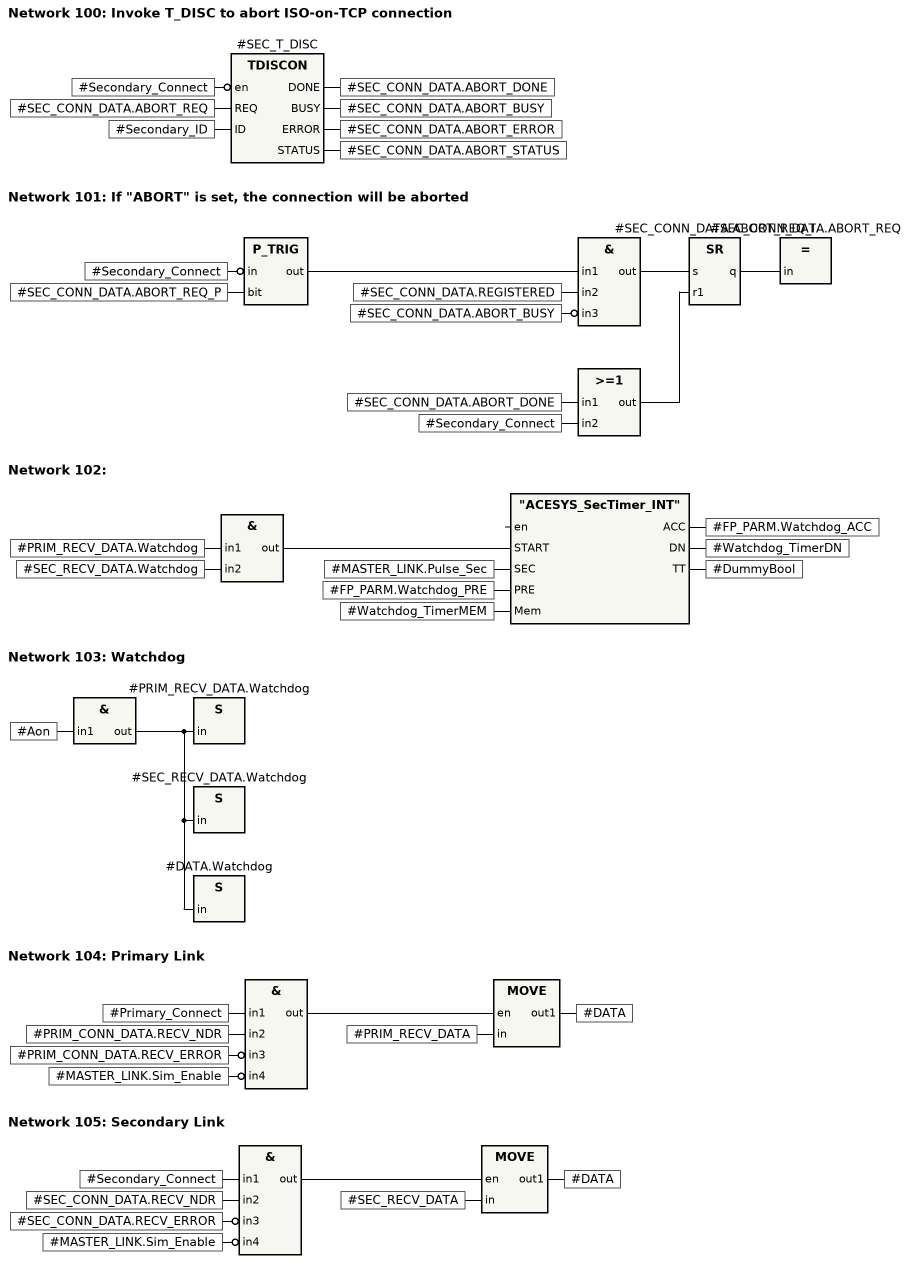
   IF NOT #Secondary_Connect THEN
       #SEC_T_DISC(REQ := #SEC_CONN_DATA.ABORT_REQ,   // TDISCON
                   ID := #Secondary_ID,
                   DONE => #SEC_CONN_DATA.ABORT_DONE,
                   BUSY => #SEC_CONN_DATA.ABORT_BUSY,
                   ERROR => #SEC_CONN_DATA.ABORT_ERROR,
                   STATUS => #SEC_CONN_DATA.ABORT_STATUS);
   END_IF;
END_REGION

REGION Network 101: If "ABORT" is set, the connection will be aborted
   #_w1 := NOT #Secondary_Connect AND NOT #SEC_CONN_DATA.ABORT_REQ_P;   // rising edge
   #SEC_CONN_DATA.ABORT_REQ_P := NOT #Secondary_Connect;
   IF #_w1 AND #SEC_CONN_DATA.REGISTERED AND NOT #SEC_CONN_DATA.ABORT_BUSY THEN
       #SEC_CONN_DATA.ABORT_REQ_I := TRUE;   // SR flip-flop
   END_IF;
   IF #SEC_CONN_DATA.ABORT_DONE OR #Secondary_Connect THEN #SEC_CONN_DATA.ABORT_REQ_I := FALSE; END_IF;
   #SEC_CONN_DATA.ABORT_REQ := #SEC_CONN_DATA.ABORT_REQ_I;
END_REGION

REGION Network 102
   "ACESYS_SecTimer_INT"(START := #PRIM_RECV_DATA.Watchdog AND #SEC_RECV_DATA.Watchdog,
                         SEC := #MASTER_LINK.Pulse_Sec,
                         PRE := #FP_PARM.Watchdog_PRE,
                         Mem := #Watchdog_TimerMEM,
                         ACC => #FP_PARM.Watchdog_ACC,
                         DN => #Watchdog_TimerDN,
                         TT => #DummyBool);
END_REGION

REGION Network 103: Watchdog
   IF #Aon THEN
       #PRIM_RECV_DATA.Watchdog := TRUE;
       #SEC_RECV_DATA.Watchdog := TRUE;
       #DATA.Watchdog := TRUE;
   END_IF;
END_REGION

REGION Network 104: Primary Link
   IF #Primary_Connect AND #PRIM_CONN_DATA.RECV_NDR AND NOT #PRIM_CONN_DATA.RECV_ERROR AND NOT #MASTER_LINK.Sim_Enable THEN
       #DATA := #PRIM_RECV_DATA;
   END_IF;
END_REGION

REGION Network 105: Secondary Link
   IF #Secondary_Connect AND #SEC_CONN_DATA.RECV_NDR AND NOT #SEC_CONN_DATA.RECV_ERROR AND NOT #MASTER_LINK.Sim_Enable THEN
       #DATA := #SEC_RECV_DATA;
   END_IF;
END_REGION

REGION Network 106: Clear Received Data if Watchdog Timer Elapsed
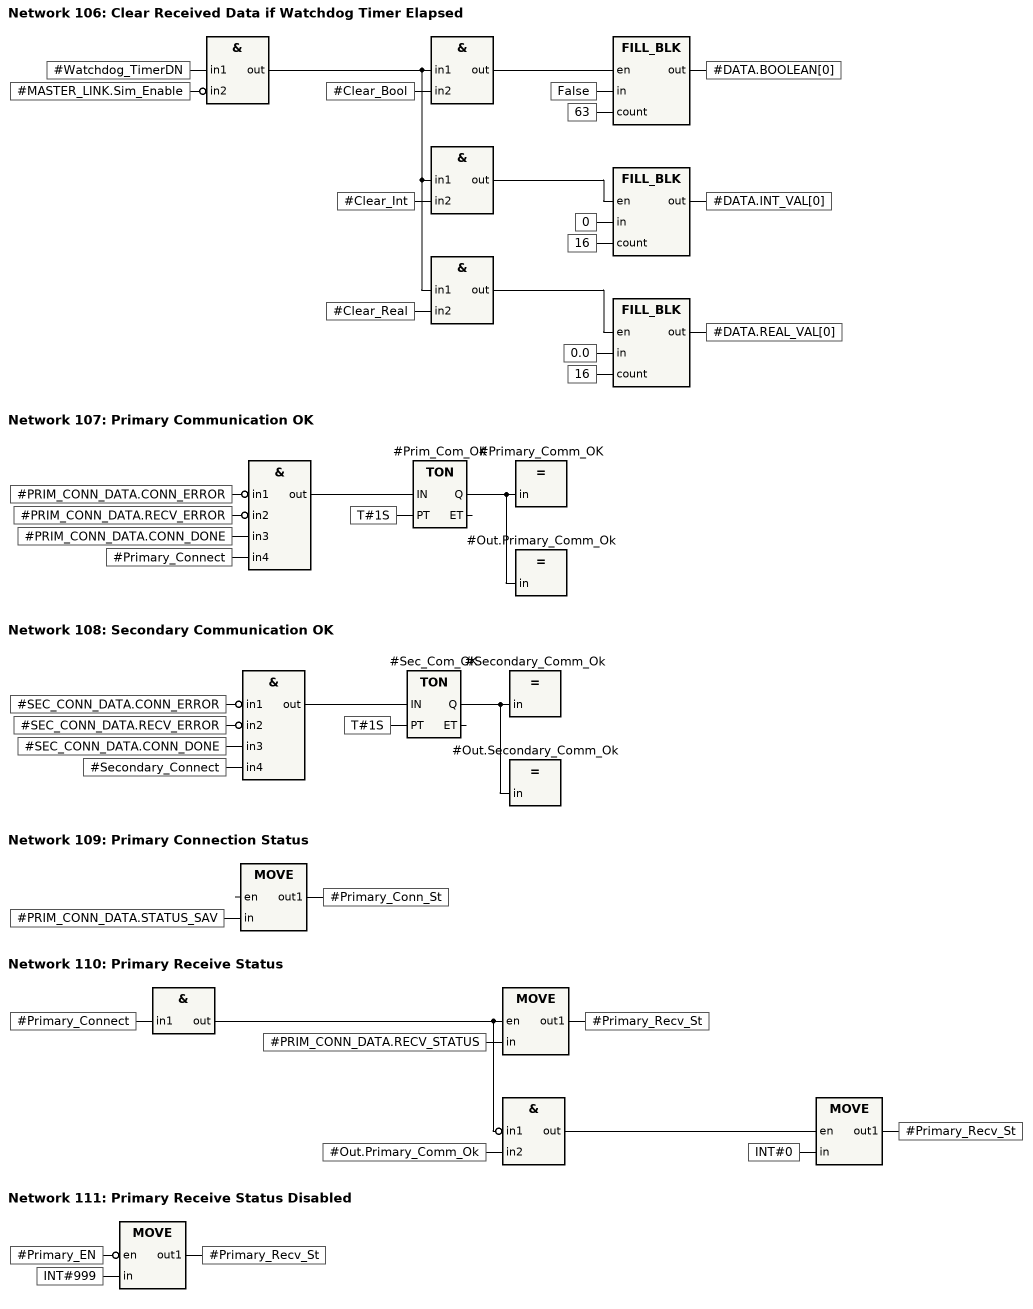
   #_w1 := #Watchdog_TimerDN AND NOT #MASTER_LINK.Sim_Enable;
   IF #_w1 AND #Clear_Bool THEN FILL_BLK(IN := False, COUNT := 63, OUT => #DATA.BOOLEAN[0]); END_IF;
   IF #_w1 AND #Clear_Int THEN FILL_BLK(IN := 0, COUNT := 16, OUT => #DATA.INT_VAL[0]); END_IF;
   IF #_w1 AND #Clear_Real THEN FILL_BLK(IN := 0.0, COUNT := 16, OUT => #DATA.REAL_VAL[0]); END_IF;
END_REGION

REGION Network 107: Primary Communication OK
   #Prim_Com_OK(IN := NOT #PRIM_CONN_DATA.CONN_ERROR AND NOT #PRIM_CONN_DATA.RECV_ERROR AND #PRIM_CONN_DATA.CONN_DONE AND #Primary_Connect,   // TON
                PT := T#1S);
   #Primary_Comm_OK := #Prim_Com_OK.Q;
   #Out.Primary_Comm_Ok := #Prim_Com_OK.Q;
END_REGION

REGION Network 108: Secondary Communication OK
   #Sec_Com_OK(IN := NOT #SEC_CONN_DATA.CONN_ERROR AND NOT #SEC_CONN_DATA.RECV_ERROR AND #SEC_CONN_DATA.CONN_DONE AND #Secondary_Connect,   // TON
               PT := T#1S);
   #Secondary_Comm_Ok := #Sec_Com_OK.Q;
   #Out.Secondary_Comm_Ok := #Sec_Com_OK.Q;
END_REGION

REGION Network 109: Primary Connection Status
   #Primary_Conn_St := #PRIM_CONN_DATA.STATUS_SAV;
END_REGION

REGION Network 110: Primary Receive Status
   IF #Primary_Connect THEN #Primary_Recv_St := #PRIM_CONN_DATA.RECV_STATUS; END_IF;
   IF NOT #Primary_Connect AND #Out.Primary_Comm_Ok THEN #Primary_Recv_St := INT#0; END_IF;
END_REGION

REGION Network 111: Primary Receive Status Disabled
   IF NOT #Primary_EN THEN #Primary_Recv_St := INT#999; END_IF;
END_REGION

REGION Network 112: Secondary Connection Status
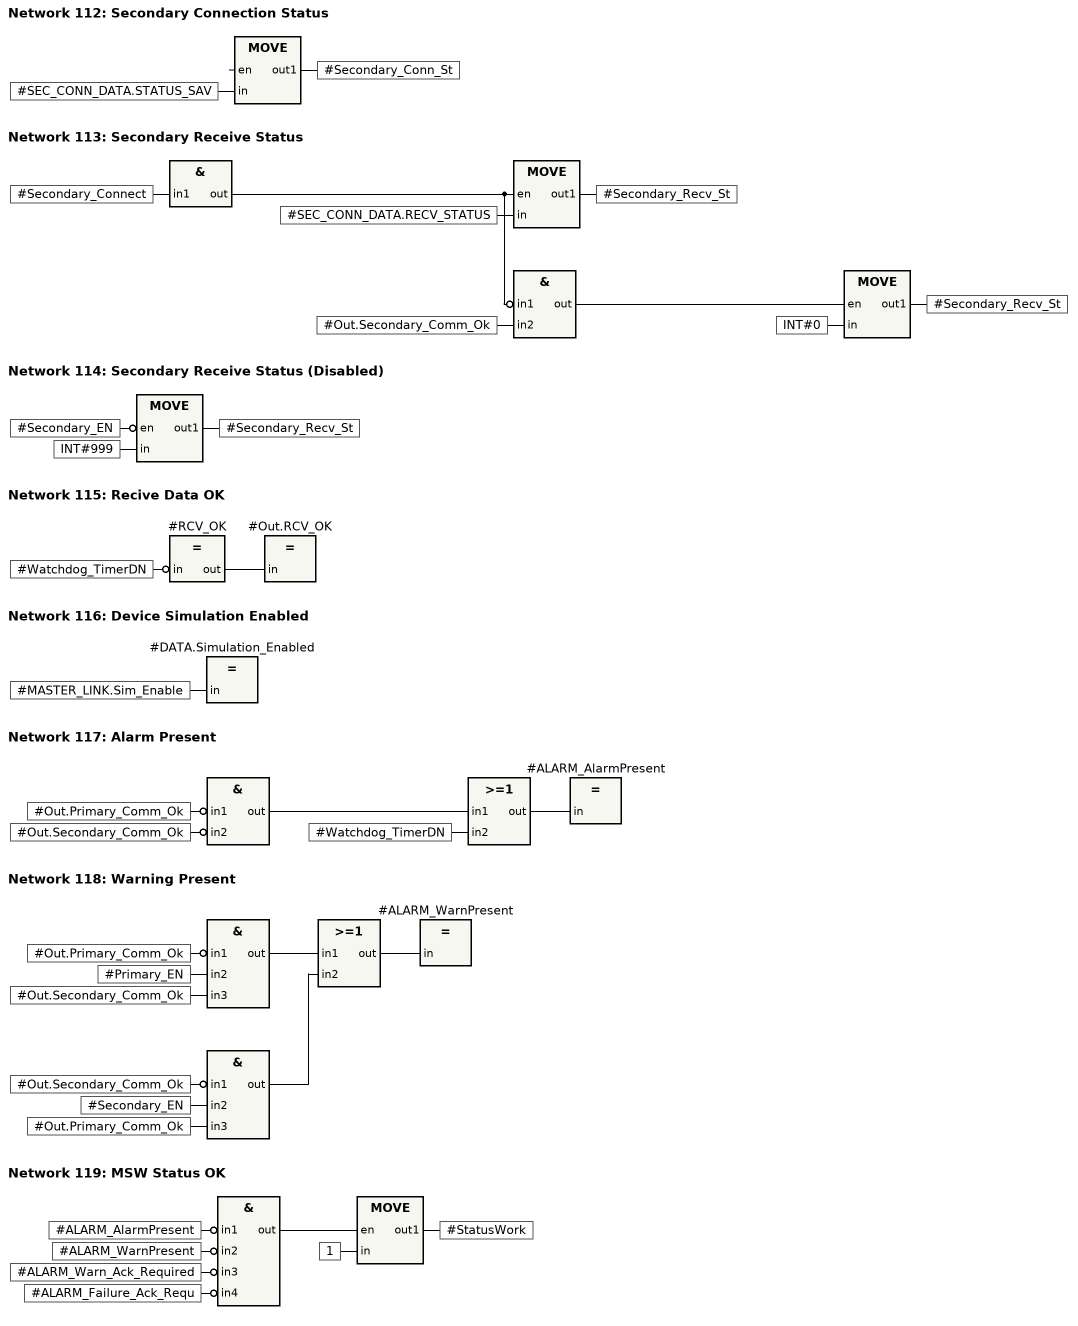
   #Secondary_Conn_St := #SEC_CONN_DATA.STATUS_SAV;
END_REGION

REGION Network 113: Secondary Receive Status
   IF #Secondary_Connect THEN #Secondary_Recv_St := #SEC_CONN_DATA.RECV_STATUS; END_IF;
   IF NOT #Secondary_Connect AND #Out.Secondary_Comm_Ok THEN #Secondary_Recv_St := INT#0; END_IF;
END_REGION

REGION Network 114: Secondary Receive Status (Disabled)
   IF NOT #Secondary_EN THEN #Secondary_Recv_St := INT#999; END_IF;
END_REGION

REGION Network 115: Recive Data OK
   #RCV_OK := NOT #Watchdog_TimerDN;
   #Out.RCV_OK := NOT #Watchdog_TimerDN;
END_REGION

REGION Network 116: Device Simulation Enabled
   // >>>>>>>Simulation Enable>>>>>>>
   #DATA.Simulation_Enabled := #MASTER_LINK.Sim_Enable;
END_REGION

REGION Network 117: Alarm Present
   #ALARM_AlarmPresent := (NOT #Out.Primary_Comm_Ok AND NOT #Out.Secondary_Comm_Ok) OR #Watchdog_TimerDN;
END_REGION

REGION Network 118: Warning Present
   #ALARM_WarnPresent := (NOT #Out.Primary_Comm_Ok AND #Primary_EN AND #Out.Secondary_Comm_Ok) OR (NOT #Out.Secondary_Comm_Ok AND #Secondary_EN AND #Out.Primary_Comm_Ok);
END_REGION

REGION Network 119: MSW Status OK
   IF NOT #ALARM_AlarmPresent AND NOT #ALARM_WarnPresent AND NOT #ALARM_Warn_Ack_Required AND NOT #ALARM_Failure_Ack_Requ THEN
       #StatusWork := 1;
   END_IF;
END_REGION

REGION Network 120: Skip = Skip Alarm
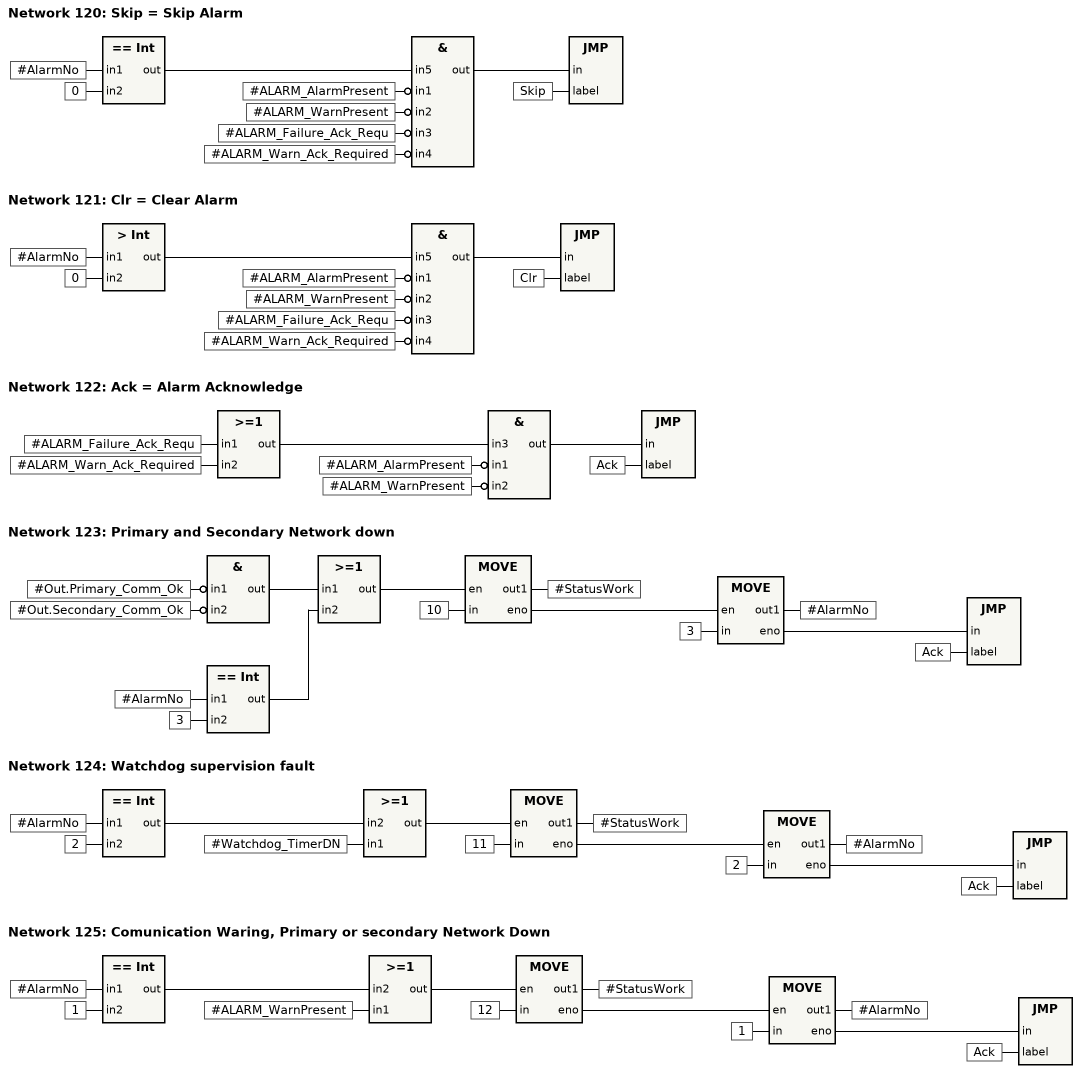
   IF (#AlarmNo = 0) AND NOT #ALARM_AlarmPresent AND NOT #ALARM_WarnPresent AND NOT #ALARM_Failure_Ack_Requ AND NOT #ALARM_Warn_Ack_Required THEN
       GOTO Skip;
   END_IF;
END_REGION

REGION Network 121: Clr = Clear Alarm
   IF (#AlarmNo > 0) AND NOT #ALARM_AlarmPresent AND NOT #ALARM_WarnPresent AND NOT #ALARM_Failure_Ack_Requ AND NOT #ALARM_Warn_Ack_Required THEN
       GOTO Clr;
   END_IF;
END_REGION

REGION Network 122: Ack = Alarm Acknowledge
   IF (#ALARM_Failure_Ack_Requ OR #ALARM_Warn_Ack_Required) AND NOT #ALARM_AlarmPresent AND NOT #ALARM_WarnPresent THEN
       GOTO Ack;
   END_IF;
END_REGION

REGION Network 123: Primary and Secondary Network down
   #_w1 := (NOT #Out.Primary_Comm_Ok AND NOT #Out.Secondary_Comm_Ok) OR (#AlarmNo = 3);
   IF #_w1 THEN
       #StatusWork := 10;
       #AlarmNo := 3;
       GOTO Ack;
   END_IF;
END_REGION

REGION Network 124: Watchdog supervision fault
   #_w1 := (#AlarmNo = 2) OR #Watchdog_TimerDN;
   IF #_w1 THEN
       #StatusWork := 11;
       #AlarmNo := 2;
       GOTO Ack;
   END_IF;
END_REGION

REGION Network 125: Comunication Waring, Primary or secondary Network Down
   #_w1 := (#AlarmNo = 1) OR #ALARM_WarnPresent;
   IF #_w1 THEN
       #StatusWork := 12;
       #AlarmNo := 1;
       GOTO Ack;
   END_IF;
END_REGION

REGION Network 126
   // >>>>>>>Alarm Acknowledge>>>>>>>
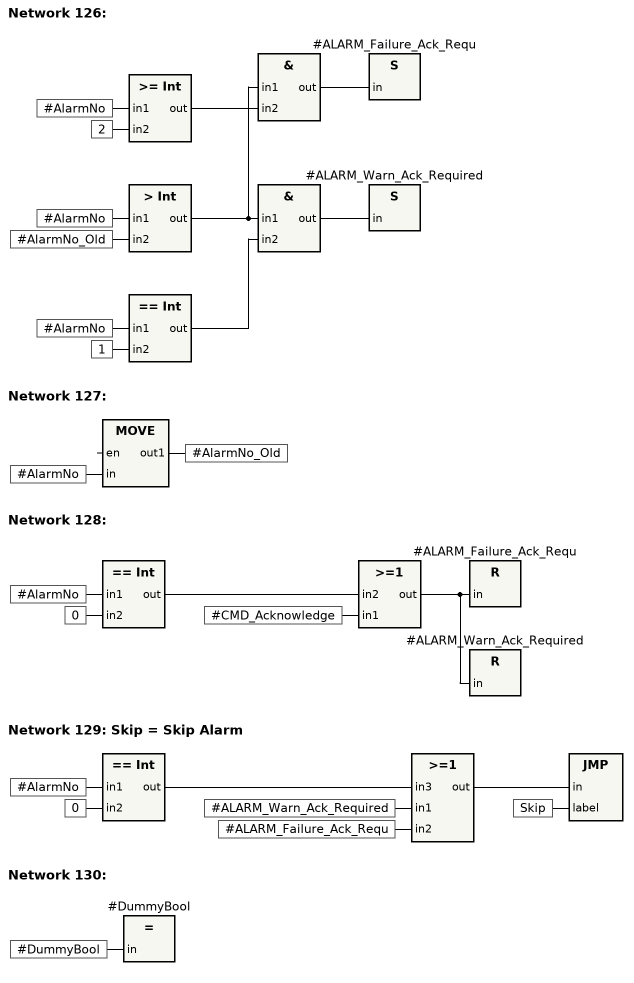
   Ack:
   #_w1 := #AlarmNo > #AlarmNo_Old;
   IF #_w1 AND (#AlarmNo >= 2) THEN #ALARM_Failure_Ack_Requ := TRUE; END_IF;
   IF #_w1 AND (#AlarmNo = 1) THEN #ALARM_Warn_Ack_Required := TRUE; END_IF;
END_REGION

REGION Network 127
   #AlarmNo_Old := #AlarmNo;
END_REGION

REGION Network 128
   IF (#AlarmNo = 0) OR #CMD_Acknowledge THEN
       #ALARM_Failure_Ack_Requ := FALSE;
       #ALARM_Warn_Ack_Required := FALSE;
   END_IF;
END_REGION

REGION Network 129: Skip = Skip Alarm
   IF (#AlarmNo = 0) OR #ALARM_Warn_Ack_Required OR #ALARM_Failure_Ack_Requ THEN GOTO Skip; END_IF;
END_REGION

REGION Network 130
   // >>>>>>>Clear Alarm>>>>>>>
   Clr:
   #DummyBool := #DummyBool;
END_REGION

REGION Network 131
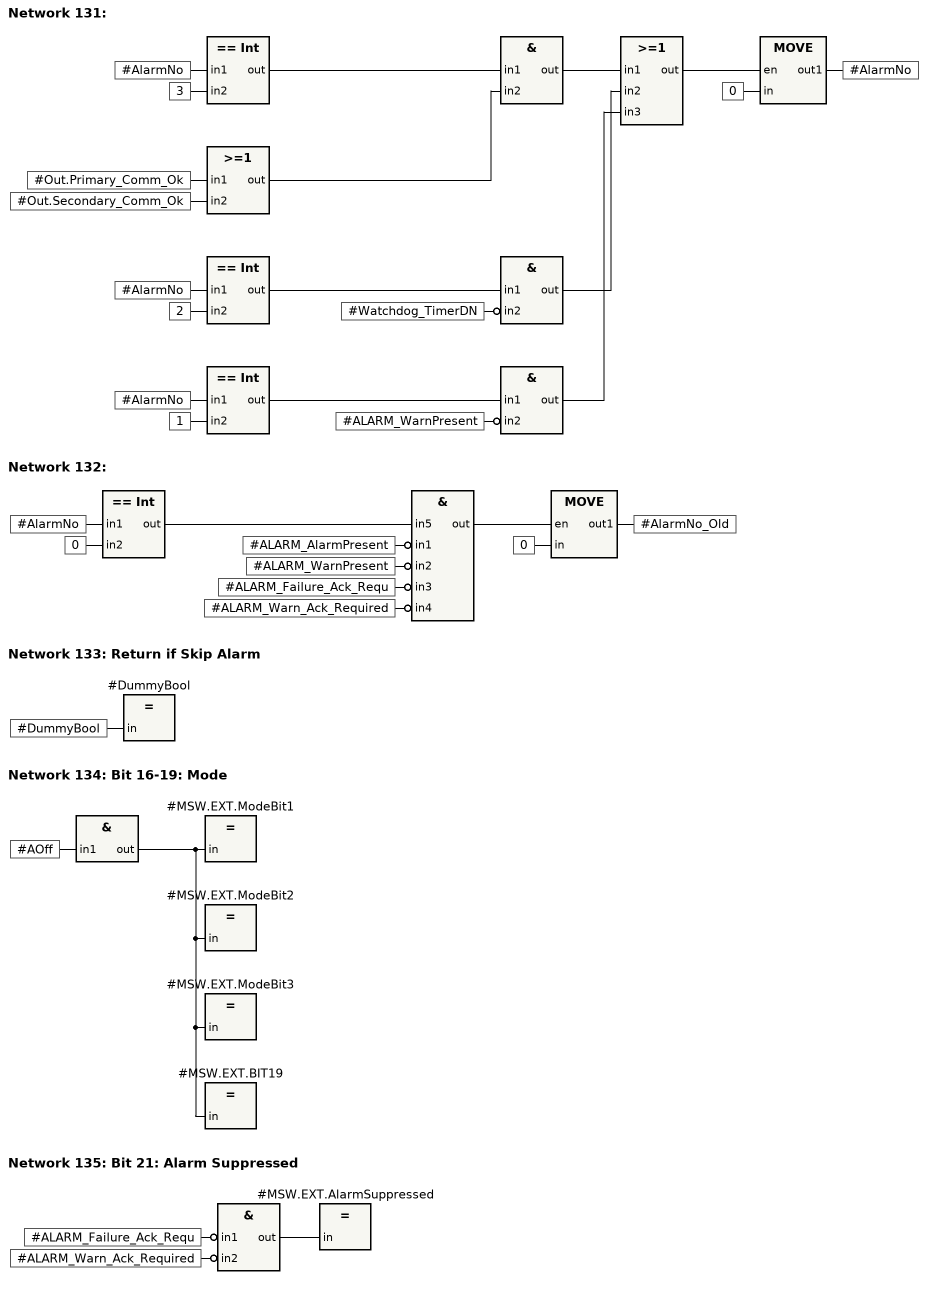
   IF ((#AlarmNo = 3) AND (#Out.Primary_Comm_Ok OR #Out.Secondary_Comm_Ok)) OR ((#AlarmNo = 2) AND NOT #Watchdog_TimerDN) OR ((#AlarmNo = 1) AND NOT #ALARM_WarnPresent) THEN
       #AlarmNo := 0;
   END_IF;
END_REGION

REGION Network 132
   IF (#AlarmNo = 0) AND NOT #ALARM_AlarmPresent AND NOT #ALARM_WarnPresent AND NOT #ALARM_Failure_Ack_Requ AND NOT #ALARM_Warn_Ack_Required THEN
       #AlarmNo_Old := 0;
   END_IF;
END_REGION

REGION Network 133: Return if Skip Alarm
   Skip:
   #DummyBool := #DummyBool;
END_REGION

REGION Network 134: Bit 16-19: Mode
   // 0 = Auto
   // 1= Single Start
   // 2 = Manual
   // 3= Local
   // 4= Test Mode
   #MSW.EXT.ModeBit1 := #AOff;
   #MSW.EXT.ModeBit2 := #AOff;
   #MSW.EXT.ModeBit3 := #AOff;
   #MSW.EXT.BIT19 := #AOff;
END_REGION

REGION Network 135: Bit 21: Alarm Suppressed
   #MSW.EXT.AlarmSuppressed := NOT #ALARM_Failure_Ack_Requ AND NOT #ALARM_Warn_Ack_Required;
END_REGION

REGION Network 136: Bit: 22 Alarm Condition Present
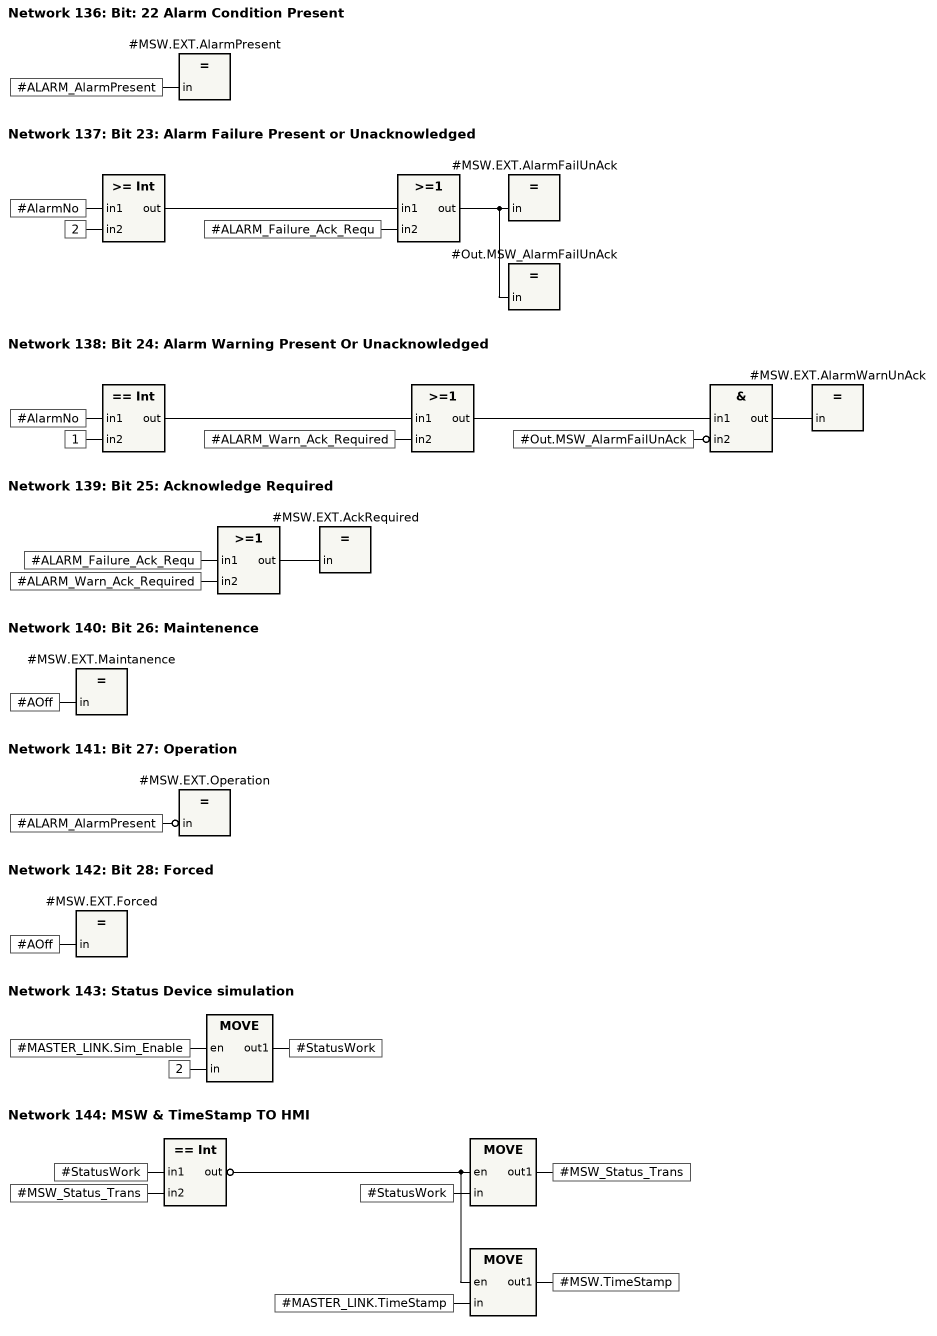
   #MSW.EXT.AlarmPresent := #ALARM_AlarmPresent;
END_REGION

REGION Network 137: Bit 23: Alarm Failure Present or Unacknowledged
   #MSW.EXT.AlarmFailUnAck := (#AlarmNo >= 2) OR #ALARM_Failure_Ack_Requ;
   #Out.MSW_AlarmFailUnAck := #MSW.EXT.AlarmFailUnAck;
END_REGION

REGION Network 138: Bit 24: Alarm Warning Present Or Unacknowledged
   #MSW.EXT.AlarmWarnUnAck := ((#AlarmNo = 1) OR #ALARM_Warn_Ack_Required) AND NOT #Out.MSW_AlarmFailUnAck;
END_REGION

REGION Network 139: Bit 25: Acknowledge Required
   #MSW.EXT.AckRequired := #ALARM_Failure_Ack_Requ OR #ALARM_Warn_Ack_Required;
END_REGION

REGION Network 140: Bit 26: Maintenence
   #MSW.EXT.Maintanence := #AOff;
END_REGION

REGION Network 141: Bit 27: Operation
   #MSW.EXT.Operation := NOT #ALARM_AlarmPresent;
END_REGION

REGION Network 142: Bit 28: Forced
   #MSW.EXT.Forced := #AOff;
END_REGION

REGION Network 143: Status Device simulation
   IF #MASTER_LINK.Sim_Enable THEN #StatusWork := 2; END_IF;
END_REGION

REGION Network 144: MSW & TimeStamp TO HMI
   #_w1 := NOT (#StatusWork = #MSW_Status_Trans);
   IF #_w1 THEN
       #MSW_Status_Trans := #StatusWork;
       #MSW.TimeStamp := #MASTER_LINK.TimeStamp;
   END_IF;
END_REGION

REGION Network 145: MSW Transfer to Actual
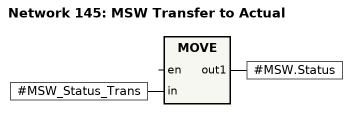
   #MSW.Status := #MSW_Status_Trans;
END_REGION
END_FUNCTION_BLOCK

FUNCTION_BLOCK "ACESYS_SEND_RECV"   // FB227, FBD
TITLE = ACESYS V8.0 - Build 001 - SEND_RECV
{ S7_Optimized_Access := 'FALSE' }
AUTHOR : FLSMIDTH
FAMILY : ACESYS
NAME : SEND_RECV
VERSION : 8.0
// PLC to PLC H Communication Block
   VAR_INPUT
      CPU00_CONN1_EN : Bool;   // S7400H CPU00 Connection 1 Enable
      CPU00_CONN2_EN : Bool;   // S7400H CPU00 Connection 2 Enable
      CPU01_CONN1_EN : Bool;   // S7400H CPU01 Connection 3 Enable
      CPU01_CONN2_EN : Bool;   // S7400H CPU01 Connection 4 Enable
      Clear_Bool : Bool;   // Clear Boolean Variables in case of Comm.Fault
      Clear_Int : Bool;   // Clear Integer Variables in case of Comm.Fault
      Clear_Real : Bool;   // Clear Real Variables in case of Comm.Fault
      Red_Setup : Bool;   // Redundancy_Configuration_Enable
      MASTER_LINK : "ACESYS_MASTER_LINK";
   END_VAR
   VAR_OUTPUT
      Communication_OK : Bool;   // Any one of The Communication OK
      SEND_OK : Bool;   // Connection Send OK
      RECV_OK : Bool;   // Connection Receive OK
      CURR_Connection : Int;   // Active Connection 1 Details
      CPU00_CONN1_Comm_OK : Bool;   // CPU00_Connection1 Communication OK
      CPU00_CONN1_Conn_St : Word;   // CPU00_Connection1 Status
      CPU00_CONN1_Send_St : Word;   // CPU00_Connection1 Send Status
      CPU00_CONN1_Recv_St : Word;   // CPU00_Connection1 Receive Status
      CPU00_CONN2_Comm_OK : Bool;   // CPU00_Connection2 Communication OK
      CPU00_CONN2_Conn_St : Word;   // CPU00_Connection2 Status
      CPU00_CONN2_Send_St : Word;   // CPU00_Connection2 Send Status
      CPU00_CONN2_Recv_St : Word;   // CPU00_Connection2 Receive Status
      CPU01_CONN1_Comm_OK : Bool;   // CPU01_Connection1 Communication OK
      CPU01_CONN1_Conn_St : Word;   // CPU01_Connection1 Status
      CPU01_CONN1_Send_St : Word;   // CPU00_Connection Send Status
      CPU01_CONN1_Recv_St : Word;   // CPU00_Connection Receive Status
      CPU01_CONN2_Comm_OK : Bool;   // CPU01_Connection2 Communication OK
      CPU01_CONN2_Conn_St : Word;   // CPU01_Connection2 Status
      CPU01_CONN2_Send_St : Word;   // CPU01_Connection2 Send Status
      CPU01_CONN2_Recv_St : Word;   // CPU01_Connection2 Receive Status
      RECV_DATA : "ACESYS_PLCToPLC_H";
      MSW : "ACESYS_HMI_STAT_32T";
   END_VAR
   VAR_IN_OUT
      Send_DATA : "ACESYS_PLCToPLC_H";
   END_VAR
   VAR
      BlockInfo : Struct
         SpareINT_15 : Int;
         SpareINT_14 : Int;
         SpareINT_13 : Int;
         SpareINT_12 : Int;
         SpareINT_11 : Int;
         SpareINT_10 : Int;
         SpareINT_9 : Int;
         SpareINT_8 : Int;
         SpareINT_7 : Int;
         SpareINT_6 : Int;
         SpareINT_5 : Int;
         SpareINT_4 : Int;
         SpareINT_3 : Int;
         SpareINT_2 : Int;
         SpareINT_1 : Int;
         SpareINT_0 : Int;
         Ace_Version : Int;   // Acesys Block Version Number
         Ace_BuildNo : Int;   // Acesys Block Build Number
         DB_Number : Int;   // Block Instance DB Number
      END_STRUCT;
      FP_CMD : Struct   // Faceplate Commands
         Spare_08 : Bool;
         Spare_09 : Bool;
         Spare_10 : Bool;
         Spare_11 : Bool;
         Spare_12 : Bool;
         Spare_13 : Bool;
         Spare_14 : Bool;
         AckAlarm : Bool;   // Alarm Acknowledge
         Spare_00 : Bool;
         Spare_01 : Bool;
         Spare_02 : Bool;
         Spare_03 : Bool;
         Spare_04 : Bool;
         Spare_05 : Bool;
         Spare_06 : Bool;
         Spare_07 : Bool;
      END_STRUCT;
      FP_PARM : Struct   // Faceplate Parameters
         Watchdog_PRE : Int := 5;   // Watchdog Time
         Watchdog_ACC : Int;   // Watchdog Time
         FREQCHANGE_MASTER_PRE : Int;
         FREQCHANGE_MASTER_ACC : Int;
         CURR_CONN : Int;   // Active Connection Details (STAT)
         H_State : Int;   // CPU In Redundancy State
         Master_Slave_Info : Int;   // CPU Master/Slave Information
         RunningCPU_Info : Int;   // CPU Running Status
      END_STRUCT;
      Conn1_Watchdog_Fault : Bool;
      Conn2_Watchdog_Fault : Bool;
      Conn3_Watchdog_Fault : Bool;
      Conn4_Watchdog_Fault : Bool;
      ONS : Struct
         H_Changeover_Mstr0 : Bool;
         H_Changeover_Mstr1 : Bool;
         H_Changeover_Mstr0_Reset : Bool;
         H_Changeover_Mstr1_Reset : Bool;
         Watchdog_Fail_P : Bool;
         Watchdog_Fail_N : Bool;
         Conn1Watchdog_Fail_P : Bool;
         Conn1Watchdog_Fail_N : Bool;
         Conn2Watchdog_Fail_P : Bool;
         Conn2Watchdog_Fail_N : Bool;
         Conn3Watchdog_Fail_P : Bool;
         Conn3Watchdog_Fail_N : Bool;
         Conn4Watchdog_Fail_P : Bool;
         Conn4Watchdog_Fail_N : Bool;
      END_STRUCT;
      CPU00_CONN1_TSEND_Migra : TSEND;
      CPU00_CONN1_TRECV_Migra : TRCV;
      CPU00_CONN1_TCONN_Migra : TCON;
      CPU00_CONN1_TDISC_Migra : TDISCON;
      CPU00_CONN1_DATA : Struct
         REGISTERED : Bool;
         CONN_DONE : Bool;
         CONN_BUSY : Bool;
         CONN_ERROR : Bool;
         CONN_SETA : Bool;
         DISCONNECT : Bool;
         CONN_STATUS : Word;
         STATUS_SAV : Int;
         SEND_REQ : Bool;
         SEND_DONE : Bool;
         SEND_BUSY : Bool;
         SEND_ERROR : Bool;
         SEND_REQ_P : Bool;
         SEND_REQ_I : Bool;
         SEND_STATUS : Word;
         ABORT_REQ : Bool;
         ABORT_DONE : Bool;
         ABORT_BUSY : Bool;
         ABORT_ERROR : Bool;
         ABORT_REQ_I : Bool;
         ABORT_REQ_P : Bool;
         ABORT_STATUS : Word;
      END_STRUCT;
      CPU00_CONN1_RECV : Struct
         REGISTERED : Bool;
         CONN_DONE : Bool;
         CONN_BUSY : Bool;
         CONN_ERROR : Bool;
         CONN_SETA : Bool;
         DISCONNECT : Bool;
         CONN_STATUS : Word;
         STATUS_SAV : Int;
         RECV_NDR : Bool;
         RECV_BUSY : Bool;
         RECV_ERROR : Bool;
         RECV_STATUS : Word;
         RECV_LEN : Int;
         RECV_LEN_S : Int;
         ABORT_REQ : Bool;
         ABORT_DONE : Bool;
         ABORT_BUSY : Bool;
         ABORT_ERROR : Bool;
         ABORT_REQ_I : Bool;
         ABORT_REQ_P : Bool;
         ABORT_STATUS : Word;
      END_STRUCT;
      CPU00_CONN1_RECV_DATA : "ACESYS_PLCToPLC_H";
      CPU00_CONN2_TSEND_Migra : TSEND;
      CPU00_CONN2_TRECV_Migra : TRCV;
      CPU00_CONN2_TCONN_Migra : TCON;
      CPU00_CONN2_TDISC_Migra : TDISCON;
      CPU00_CONN2_DATA : Struct
         REGISTERED : Bool;
         CONN_DONE : Bool;
         CONN_BUSY : Bool;
         CONN_ERROR : Bool;
         CONN_SETA : Bool;
         DISCONNECT : Bool;
         CONN_STATUS : Word;
         STATUS_SAV : Int;
         SEND_REQ : Bool;
         SEND_DONE : Bool;
         SEND_BUSY : Bool;
         SEND_ERROR : Bool;
         SEND_REQ_P : Bool;
         SEND_REQ_I : Bool;
         SEND_STATUS : Word;
         ABORT_REQ : Bool;
         ABORT_DONE : Bool;
         ABORT_BUSY : Bool;
         ABORT_ERROR : Bool;
         ABORT_REQ_I : Bool;
         ABORT_REQ_P : Bool;
         ABORT_STATUS : Word;
      END_STRUCT;
      CPU00_CONN2_RECV : Struct
         REGISTERED : Bool;
         CONN_DONE : Bool;
         CONN_BUSY : Bool;
         CONN_ERROR : Bool;
         CONN_SETA : Bool;
         DISCONNECT : Bool;
         CONN_STATUS : Word;
         STATUS_SAV : Int;
         RECV_NDR : Bool;
         RECV_BUSY : Bool;
         RECV_ERROR : Bool;
         RECV_STATUS : Word;
         RECV_LEN : Int;
         RECV_LEN_S : Int;
         ABORT_REQ : Bool;
         ABORT_DONE : Bool;
         ABORT_BUSY : Bool;
         ABORT_ERROR : Bool;
         ABORT_REQ_I : Bool;
         ABORT_REQ_P : Bool;
         ABORT_STATUS : Word;
      END_STRUCT;
      CPU00_CONN2_RECV_DATA : "ACESYS_PLCToPLC_H";
      CPU01_CONN1_TSEND_Migra : TSEND;
      CPU01_CONN1_TRECV_Migra : TRCV;
      CPU01_CONN1_TCONN_Migra : TCON;
      CPU01_CONN1_TDISC_Migra : TDISCON;
      CPU01_CONN1_DATA : Struct
         REGISTERED : Bool;
         CONN_DONE : Bool;
         CONN_BUSY : Bool;
         CONN_ERROR : Bool;
         CONN_SETA : Bool;
         DISCONNECT : Bool;
         CONN_STATUS : Word;
         STATUS_SAV : Int;
         SEND_REQ : Bool;
         SEND_DONE : Bool;
         SEND_BUSY : Bool;
         SEND_ERROR : Bool;
         SEND_REQ_P : Bool;
         SEND_REQ_I : Bool;
         SEND_STATUS : Word;
         ABORT_REQ : Bool;
         ABORT_DONE : Bool;
         ABORT_BUSY : Bool;
         ABORT_ERROR : Bool;
         ABORT_REQ_I : Bool;
         ABORT_REQ_P : Bool;
         ABORT_STATUS : Word;
      END_STRUCT;
      CPU01_CONN1_RECV : Struct
         REGISTERED : Bool;
         CONN_DONE : Bool;
         CONN_BUSY : Bool;
         CONN_ERROR : Bool;
         CONN_SETA : Bool;
         DISCONNECT : Bool;
         CONN_STATUS : Word;
         STATUS_SAV : Int;
         RECV_NDR : Bool;
         RECV_BUSY : Bool;
         RECV_ERROR : Bool;
         RECV_STATUS : Word;
         RECV_LEN : Int;
         RECV_LEN_S : Int;
         ABORT_REQ : Bool;
         ABORT_DONE : Bool;
         ABORT_BUSY : Bool;
         ABORT_ERROR : Bool;
         ABORT_REQ_I : Bool;
         ABORT_REQ_P : Bool;
         ABORT_STATUS : Word;
      END_STRUCT;
      CPU01_CONN1_RECV_DATA : "ACESYS_PLCToPLC_H";
      CPU01_CONN2_TSEND_Migra : TSEND;
      CPU01_CONN2_TRECV_Migra : TRCV;
      CPU01_CONN2_TCONN_Migra : TCON;
      CPU01_CONN2_TDISC_Migra : TDISCON;
      CPU01_CONN2_DATA : Struct
         REGISTERED : Bool;
         CONN_DONE : Bool;
         CONN_BUSY : Bool;
         CONN_ERROR : Bool;
         CONN_SETA : Bool;
         DISCONNECT : Bool;
         CONN_STATUS : Word;
         STATUS_SAV : Int;
         SEND_REQ : Bool;
         SEND_DONE : Bool;
         SEND_BUSY : Bool;
         SEND_ERROR : Bool;
         SEND_REQ_P : Bool;
         SEND_REQ_I : Bool;
         SEND_STATUS : Word;
         ABORT_REQ : Bool;
         ABORT_DONE : Bool;
         ABORT_BUSY : Bool;
         ABORT_ERROR : Bool;
         ABORT_REQ_I : Bool;
         ABORT_REQ_P : Bool;
         ABORT_STATUS : Word;
      END_STRUCT;
      CPU01_CONN2_RECV : Struct
         REGISTERED : Bool;
         CONN_DONE : Bool;
         CONN_BUSY : Bool;
         CONN_ERROR : Bool;
         CONN_SETA : Bool;
         DISCONNECT : Bool;
         CONN_STATUS : Word;
         STATUS_SAV : Int;
         RECV_NDR : Bool;
         RECV_BUSY : Bool;
         RECV_ERROR : Bool;
         RECV_STATUS : Word;
         RECV_LEN : Int;
         RECV_LEN_S : Int;
         ABORT_REQ : Bool;
         ABORT_DONE : Bool;
         ABORT_BUSY : Bool;
         ABORT_ERROR : Bool;
         ABORT_REQ_I : Bool;
         ABORT_REQ_P : Bool;
         ABORT_STATUS : Word;
      END_STRUCT;
      CPU01_CONN2_RECV_DATA : "ACESYS_PLCToPLC_H";
      SEND_DATA_STAT_VAR : "ACESYS_PLCToPLC_H";
      CPU00_CONN1 : "ACESYS_ISO_On_TCP_TSAP";
      CPU00_CONN2 : "ACESYS_ISO_On_TCP_TSAP";
      CPU01_CONN1 : "ACESYS_ISO_On_TCP_TSAP";
      CPU01_CONN2 : "ACESYS_ISO_On_TCP_TSAP";
      TSAP16 : String[16];
      DummyString : String[16];
      Watchdog_TimerMEM : Int;
      FREQ_MSTR_CHNG_TmrMEM : Int;
      StatusWork : Int;
      AlarmNo : Int;
      AlarmNo_Old : Int;
      CMD_Acknowledge : Bool;   // Internal Acknowledge
      CONN1_INIT_COM : Bool;
      CONN2_INIT_COM : Bool;
      CONN3_INIT_COM : Bool;
      CONN4_INIT_COM : Bool;
      CONN1_En_ONS : Bool;
      CONN2_En_ONS : Bool;
      CONN3_En_ONS : Bool;
      CONN4_En_ONS : Bool;
      CONN1_Enabled_ONS : Bool;
      CONN2_Enabled_ONS : Bool;
      CONN3_Enabled_ONS : Bool;
      CONN4_Enabled_ONS : Bool;
      SPECIFIED : Bool;
      Watchdog_TimerDN : Bool;
      CONN1Watchdog_TMRDN : Bool;
      CONN2Watchdog_TMRDN : Bool;
      CONN3Watchdog_TMRDN : Bool;
      CONN4Watchdog_TMRDN : Bool;
      CONN1_ReCon_Active : Bool;   // Reconection Acive
      CONN2_ReCon_Active : Bool;   // Reconection Acive
      CONN3_ReCon_Active : Bool;   // Reconection Acive
      CONN4_ReCon_Active : Bool;   // Reconection Acive
      CONN1_SendReq_Dn : Bool;
      CONN2_SendReq_Dn : Bool;
      CONN3_SendReq_Dn : Bool;
      CONN4_SendReq_Dn : Bool;
      ALARM_AlarmPresent : Bool;
      ALARM_WarnPresent : Bool;
      ALARM_Failure_Ack_Requ : Bool;
      ALARM_Warn_Ack_Required : Bool;
      CONN1_Connect : Bool;   // Conect Primary Link
      CONN2_Connect : Bool;   // Conect Secondary Link
      CONN3_Connect : Bool;   // Conect Primary Link
      CONN4_Connect : Bool;   // Conect Secondary Link
      CPU00_CONN1_Enable : Bool;
      CPU00_CONN2_Enable : Bool;
      CPU01_CONN1_Enable : Bool;
      CPU01_CONN2_Enable : Bool;
      Freq_Change_MSTR0_DN : Bool;
      Freq_Change_MSTR1_DN : Bool;
      Conn1_Trigger : Bool;   // Default Connection
      Conn2_Trigger : Bool;
      Conn3_Trigger : Bool;
      Conn4_Trigger : Bool;
      CPU0CONN1_ComOK_Stat : Bool;
      CPU0CONN2_ComOK_Stat : Bool;
      CPU1CONN1_ComOK_Stat : Bool;
      CPU1CONN2_ComOK_Stat : Bool;
      MSWEXTAlarmFailUnAckStat : Bool;
      Spare_Bool_05 : Bool;
      Spare_Bool_04 : Bool;
      H_ChangeMastr0 : Bool;
      H_ChangeMastr1 : Bool;
      Spare_Bool_03 : Bool;
      Spare_Bool_02 : Bool;
      Spare_Bool_01 : Bool;
      Conn1Watchdog_TimerMEM : Int;
      Conn2Watchdog_TimerMEM : Int;
      Conn3Watchdog_TimerMEM : Int;
      Conn4Watchdog_TimerMEM : Int;
      Conn1_Watchdog_ACC : Int;
      Conn2_Watchdog_ACC : Int;
      Conn3_Watchdog_ACC : Int;
      Conn4_Watchdog_ACC : Int;
      Freq_MSTR_00_ACC : Int;
      Freq_MSTR_01_ACC : Int;
      Freq_MSTR_00_Mem : Int;
      Freq_MSTR_01_Mem : Int;
      Conn4_Send_Freq_TIME : Time;
      Conn3_Send_Freq_TIME : Time;
      Conn2_Send_Freq_TIME : Time;
      Conn1_Send_Freq_TIME : Time;
      Spare_Real_3 : Real;
      Spare_Real_2 : Real;
      Spare_Real_1 : Real;
      Conn1_Send_PRE : Int;
      Conn2_Send_PRE : Int;
      Conn3_Send_PRE : Int;
      Conn4_Send_PRE : Int;
      MSW_Status_Trans : Int;
      RECV_DATA_STAT : "ACESYS_PLCToPLC_H";
      CONN1_Del_ReCon : TON_TIME;   // Delay Before Auto ReCone
      CONN1_Con_TMR : TON_TIME;
      CONN2_Del_ReCon : TON_TIME;   // Delay Before Auto ReConect
      CONN2_Con_TMR : TON_TIME;
      CONN3_Del_ReCon : TON_TIME;   // Delay Before Auto ReCone
      CONN3_Con_TMR : TON_TIME;
      CONN4_Del_ReCon : TON_TIME;   // Delay Before Auto ReConect
      CONN4_Con_TMR : TON_TIME;
      CONN1_Com_OK : TON_TIME;
      CONN2_Com_OK : TON_TIME;
      CONN3_Com_OK : TON_TIME;
      CONN4_Com_OK : TON_TIME;
      CONN1_SendDelay : TON_TIME;
      CONN2_SendDelay : TON_TIME;
      CONN3_SendDelay : TON_TIME;
      CONN4_SendDelay : TON_TIME;
      SEND_OK_TMR : TON_TIME;
   END_VAR
   VAR_TEMP
      Aon : Bool;
      AOff : Bool;
      DummyBool : Bool;
      LOC_LEN : Int;
      REM_LEN : Int;
      TMP_INT : Int;
      LOC_RS : Int;
      TMP_RS : Int;
      TMP_DEV : Int;
      DummyDInt : DInt;
      RET : Int;
      Conn1_UDT_Length : Int;
      Conn2_UDT_Length : Int;
      Conn3_UDT_Length : Int;
      Conn4_UDT_Length : Int;
      t_Zero : Int;
      PLC2PLCH_Pntr : Struct
         DB_Number : Word;
         Offset_Address : DWord;
      END_STRUCT;
      PLC2PLCH_Pointer : ANY;
      PLC2PLCH_AR1 : DWord;
      PLC2PLCH_AR2 : DWord;
      TPLC2PLCH_Pntr : Struct
         DB_Number : Word;
         Offset_Address : DWord;
      END_STRUCT;
      Connection1_Pointer : ANY;
      Connection2_Pointer : ANY;
      Connection3_Pointer : ANY;
      Connection4_Pointer : ANY;
      Connection1_Pointer_AR1 : DWord;
      Connection2_Pointer_AR1 : DWord;
      Connection3_Pointer_AR1 : DWord;
      Connection4_Pointer_AR1 : DWord;
      DummyInt : Int;
   END_VAR
   VAR_TEMP   // added for the SCL form of the ladder/FBD networks
      _w1 : Bool;
      _w2 : Bool;
   END_VAR
BEGIN

REGION Network 1: Alwayse On Bit
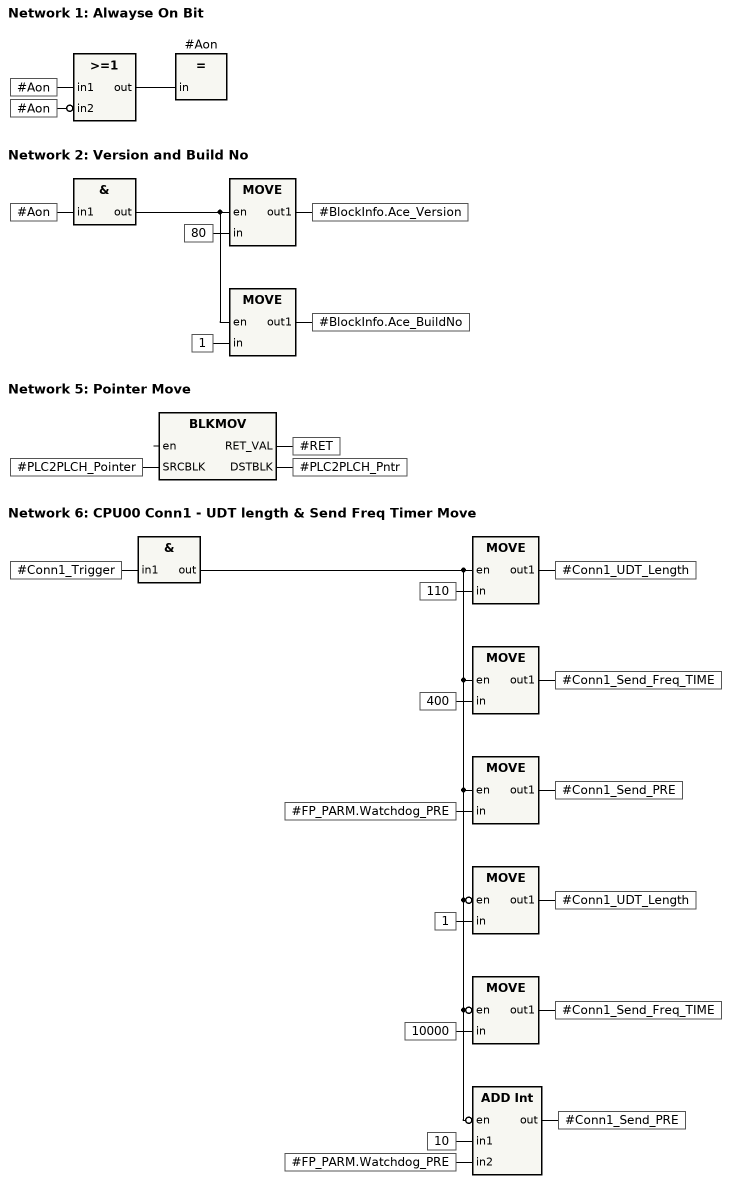
   #Aon := #Aon OR NOT #Aon;
END_REGION

REGION Network 2: Version and Build No
   IF #Aon THEN
       #BlockInfo.Ace_Version := 80;
       #BlockInfo.Ace_BuildNo := 1;
   END_IF;
END_REGION

REGION Network 3 (STL): Instance DB Number to Faceplate
         L     DINO;
         T     #BlockInfo.DB_Number;
END_REGION

REGION Network 4 (STL): Define a Pointer for the PLC2PLC H UDT in IN/OUT
   // >> Length of Pointer has to be the total Size of the UDT227 in BYTE<<

         TAR1  #PLC2PLCH_AR1;

         LAR1;

         L     16#10;  //Syntax ID
         T     LB[AR1, P#0.0];

         L     16#02;  //Data Type = Byte
         T     LB[AR1, P#1.0];

         L     6;  //Length
         T     LW[AR1, P#2.0];

         L     #BlockInfo.DB_Number;  //Area = DB
         T     LW[AR1, P#4.0];

         L     162;

         SLD   3;
         OD    16#8400_0000;
         T     LD[AR1, P#6.0];

         NOP   0;

         LAR1  #PLC2PLCH_AR1;
END_REGION

REGION Network 5: Pointer Move
   #RET := BLKMOV(SRCBLK := #PLC2PLCH_Pointer, DSTBLK => #PLC2PLCH_Pntr);
END_REGION

REGION Network 6: CPU00 Conn1 - UDT length & Send Freq Timer Move
   IF #Conn1_Trigger THEN
       #Conn1_UDT_Length := 110;
       #Conn1_Send_Freq_TIME := 400;
       #Conn1_Send_PRE := #FP_PARM.Watchdog_PRE;
   END_IF;
   IF NOT #Conn1_Trigger THEN
       #Conn1_UDT_Length := 1;
       #Conn1_Send_Freq_TIME := 10000;
       #Conn1_Send_PRE := 10 + #FP_PARM.Watchdog_PRE;
   END_IF;
END_REGION

REGION Network 7 (STL): Define a Pointer for the PLC2PLCH UDT in IN/OUT
   // >> Length of Pointer has to be the total Size of the UDT227 in BYTE<<

         TAR1  #Connection1_Pointer_AR1;

         LAR1;

         L     16#10;  //Syntax ID
         T     LB[AR1, P#0.0];

         L     16#02;  //Data Type = Byte
         T     LB[AR1, P#1.0];

         L     #Conn1_UDT_Length;  //Length
         T     LW[AR1, P#2.0];

         L     #PLC2PLCH_Pntr.DB_Number;  //Area = DB
         T     LW[AR1, P#4.0];

         L     #PLC2PLCH_Pntr.Offset_Address;

         OD    16#8400_0000;
         T     LD[AR1, P#6.0];

         NOP   0;

         LAR1  #Connection1_Pointer_AR1;
END_REGION

REGION Network 8: CPU00 Conn2 - UDT length & Send Freq Timer Move
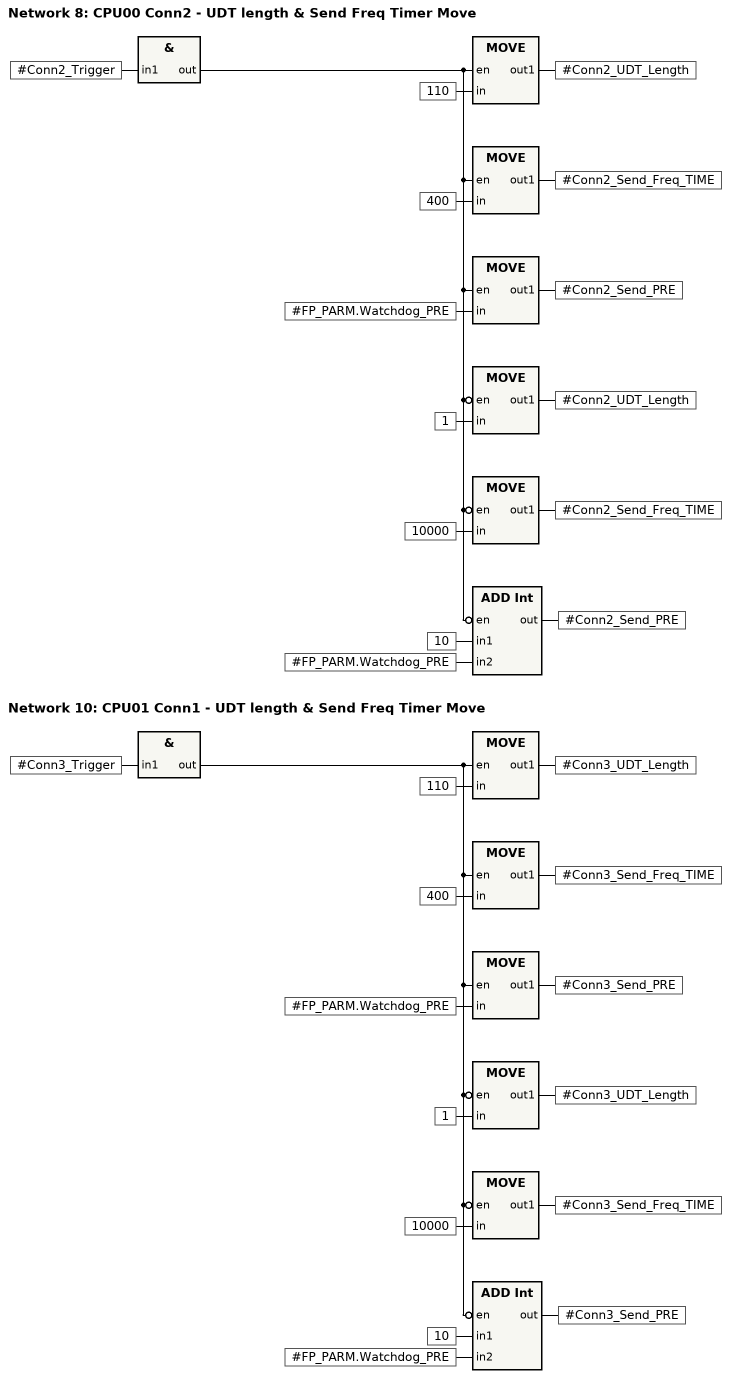
   IF #Conn2_Trigger THEN
       #Conn2_UDT_Length := 110;
       #Conn2_Send_Freq_TIME := 400;
       #Conn2_Send_PRE := #FP_PARM.Watchdog_PRE;
   END_IF;
   IF NOT #Conn2_Trigger THEN
       #Conn2_UDT_Length := 1;
       #Conn2_Send_Freq_TIME := 10000;
       #Conn2_Send_PRE := 10 + #FP_PARM.Watchdog_PRE;
   END_IF;
END_REGION

REGION Network 9 (STL): Define a Pointer for the PLC2PLCH UDT in IN/OUT
   // >> Length of Pointer has to be the total Size of the UDT227 in BYTE<<

         TAR1  #Connection2_Pointer_AR1;

         LAR1;

         L     16#10;  //Syntax ID
         T     LB[AR1, P#0.0];

         L     16#02;  //Data Type = Byte
         T     LB[AR1, P#1.0];

         L     #Conn2_UDT_Length;  //Length
         T     LW[AR1, P#2.0];

         L     #PLC2PLCH_Pntr.DB_Number;  //Area = DB
         T     LW[AR1, P#4.0];

         L     #PLC2PLCH_Pntr.Offset_Address;

         OD    16#8400_0000;
         T     LD[AR1, P#6.0];

         NOP   0;

         LAR1  #Connection2_Pointer_AR1;
END_REGION

REGION Network 10: CPU01 Conn1 - UDT length & Send Freq Timer Move
   IF #Conn3_Trigger THEN
       #Conn3_UDT_Length := 110;
       #Conn3_Send_Freq_TIME := 400;
       #Conn3_Send_PRE := #FP_PARM.Watchdog_PRE;
   END_IF;
   IF NOT #Conn3_Trigger THEN
       #Conn3_UDT_Length := 1;
       #Conn3_Send_Freq_TIME := 10000;
       #Conn3_Send_PRE := 10 + #FP_PARM.Watchdog_PRE;
   END_IF;
END_REGION

REGION Network 11 (STL): Define a Pointer for the PLC2PLCH UDT in IN/OUT
   // >> Length of Pointer has to be the total Size of the UDT227 in BYTE<<

         TAR1  #Connection3_Pointer_AR1;

         LAR1;

         L     16#10;  //Syntax ID
         T     LB[AR1, P#0.0];

         L     16#02;  //Data Type = Byte
         T     LB[AR1, P#1.0];

         L     #Conn3_UDT_Length;  //Length
         T     LW[AR1, P#2.0];

         L     #PLC2PLCH_Pntr.DB_Number;  //Area = DB
         T     LW[AR1, P#4.0];

         L     #PLC2PLCH_Pntr.Offset_Address;

         OD    16#8400_0000;
         T     LD[AR1, P#6.0];

         NOP   0;

         LAR1  #Connection3_Pointer_AR1;
END_REGION

REGION Network 12: CPU01 Conn2 - UDT length & Send Freq Timer Move
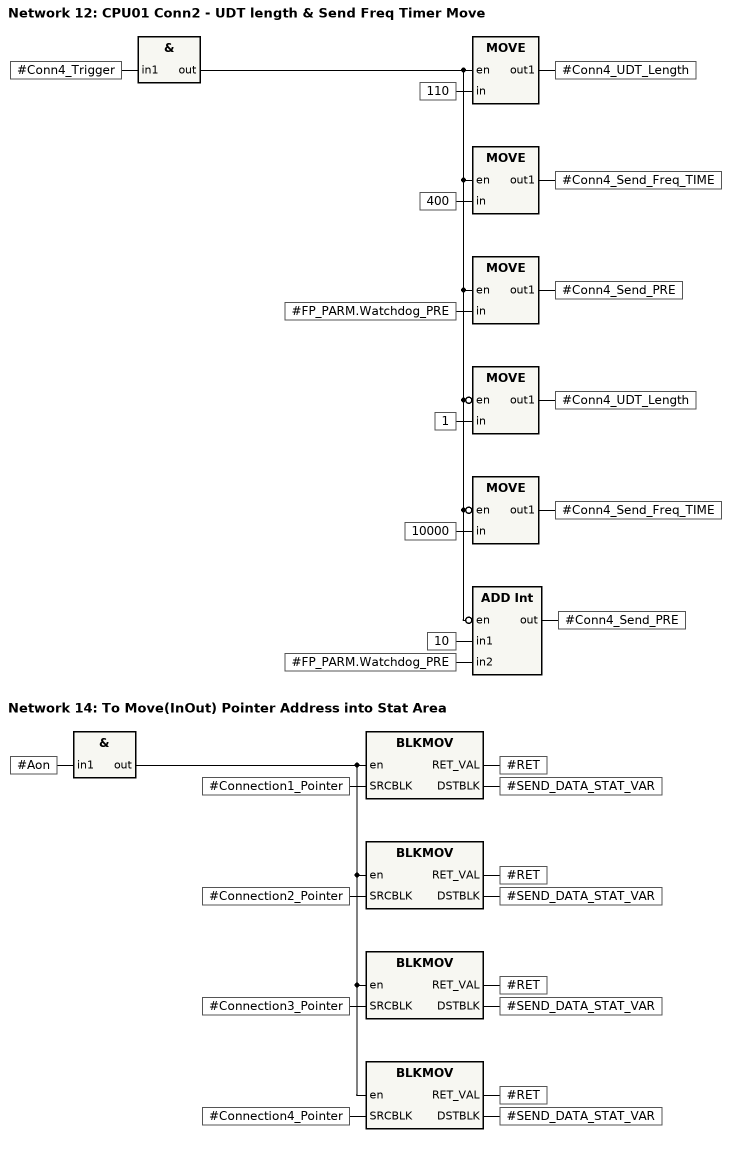
   IF #Conn4_Trigger THEN
       #Conn4_UDT_Length := 110;
       #Conn4_Send_Freq_TIME := 400;
       #Conn4_Send_PRE := #FP_PARM.Watchdog_PRE;
   END_IF;
   IF NOT #Conn4_Trigger THEN
       #Conn4_UDT_Length := 1;
       #Conn4_Send_Freq_TIME := 10000;
       #Conn4_Send_PRE := 10 + #FP_PARM.Watchdog_PRE;
   END_IF;
END_REGION

REGION Network 13 (STL): Define a Pointer for the PLC2PLCH UDT in IN/OUT
   // >> Length of Pointer has to be the total Size of the UDT226 in BYTE<<

         TAR1  #Connection4_Pointer_AR1;

         LAR1;

         L     16#10;  //Syntax ID
         T     LB[AR1, P#0.0];

         L     16#02;  //Data Type = Byte
         T     LB[AR1, P#1.0];

         L     #Conn4_UDT_Length;  //Length
         T     LW[AR1, P#2.0];

         L     #PLC2PLCH_Pntr.DB_Number;  //Area = DB
         T     LW[AR1, P#4.0];

         L     #PLC2PLCH_Pntr.Offset_Address;

         OD    16#8400_0000;
         T     LD[AR1, P#6.0];

         NOP   0;

         LAR1  #Connection4_Pointer_AR1;
END_REGION

REGION Network 14: To Move(InOut) Pointer Address into Stat Area
   IF #Aon THEN
       #RET := BLKMOV(SRCBLK := #Connection1_Pointer, DSTBLK => #SEND_DATA_STAT_VAR);
       #RET := BLKMOV(SRCBLK := #Connection2_Pointer, DSTBLK => #SEND_DATA_STAT_VAR);
       #RET := BLKMOV(SRCBLK := #Connection3_Pointer, DSTBLK => #SEND_DATA_STAT_VAR);
       #RET := BLKMOV(SRCBLK := #Connection4_Pointer, DSTBLK => #SEND_DATA_STAT_VAR);
   END_IF;
END_REGION

REGION Network 15: Calling Connection TCON Parameter FB's
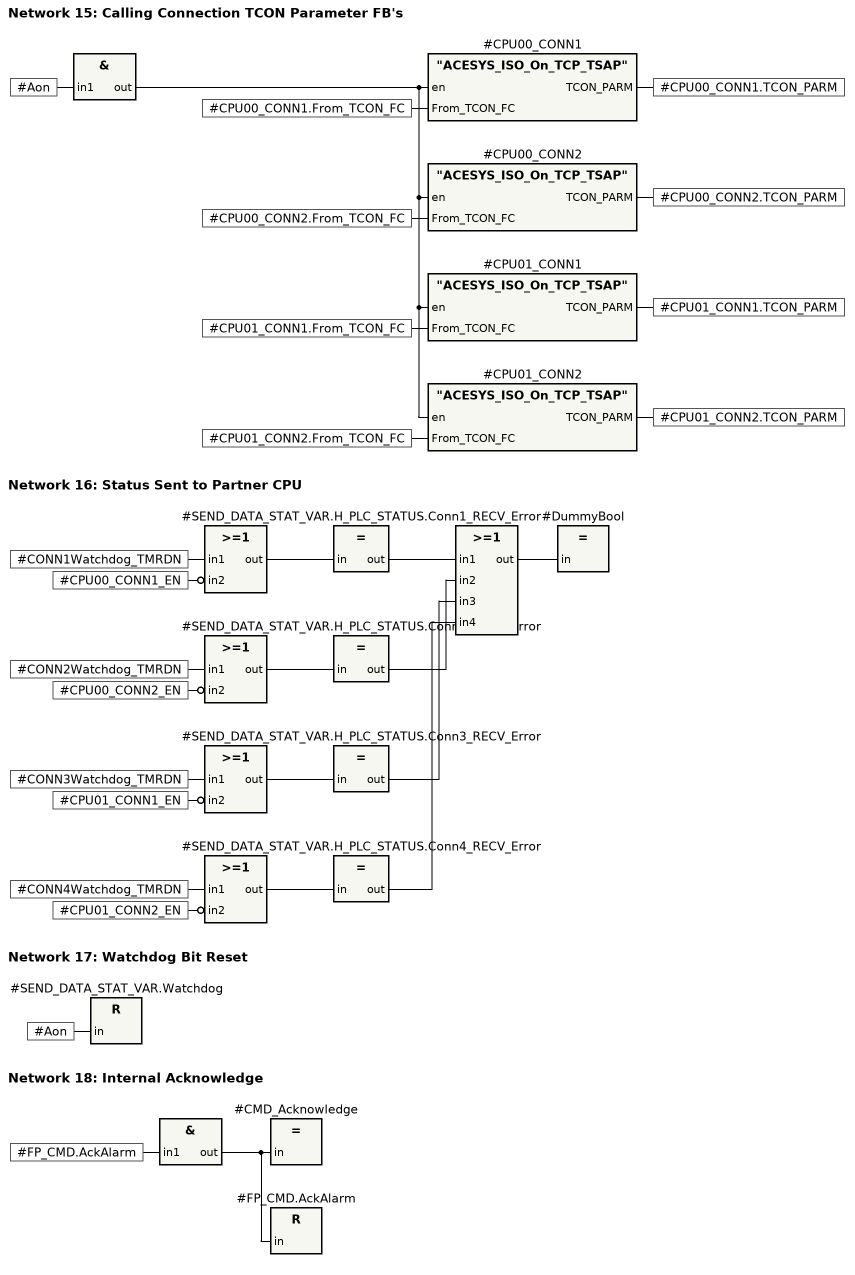
   IF #Aon THEN
       #CPU00_CONN1(From_TCON_FC := #CPU00_CONN1.From_TCON_FC, TCON_PARM => #CPU00_CONN1.TCON_PARM);   // "ACESYS_ISO_On_TCP_TSAP"
       #CPU00_CONN2(From_TCON_FC := #CPU00_CONN2.From_TCON_FC, TCON_PARM => #CPU00_CONN2.TCON_PARM);   // "ACESYS_ISO_On_TCP_TSAP"
       #CPU01_CONN1(From_TCON_FC := #CPU01_CONN1.From_TCON_FC, TCON_PARM => #CPU01_CONN1.TCON_PARM);   // "ACESYS_ISO_On_TCP_TSAP"
       #CPU01_CONN2(From_TCON_FC := #CPU01_CONN2.From_TCON_FC, TCON_PARM => #CPU01_CONN2.TCON_PARM);   // "ACESYS_ISO_On_TCP_TSAP"
   END_IF;
END_REGION

REGION Network 16: Status Sent to Partner CPU
   #SEND_DATA_STAT_VAR.H_PLC_STATUS.Conn1_RECV_Error := #CONN1Watchdog_TMRDN OR NOT #CPU00_CONN1_EN;
   #SEND_DATA_STAT_VAR.H_PLC_STATUS.Conn2_RECV_Error := #CONN2Watchdog_TMRDN OR NOT #CPU00_CONN2_EN;
   #SEND_DATA_STAT_VAR.H_PLC_STATUS.Conn3_RECV_Error := #CONN3Watchdog_TMRDN OR NOT #CPU01_CONN1_EN;
   #SEND_DATA_STAT_VAR.H_PLC_STATUS.Conn4_RECV_Error := #CONN4Watchdog_TMRDN OR NOT #CPU01_CONN2_EN;
   #DummyBool := #SEND_DATA_STAT_VAR.H_PLC_STATUS.Conn1_RECV_Error OR #SEND_DATA_STAT_VAR.H_PLC_STATUS.Conn2_RECV_Error OR #SEND_DATA_STAT_VAR.H_PLC_STATUS.Conn3_RECV_Error OR #SEND_DATA_STAT_VAR.H_PLC_STATUS.Conn4_RECV_Error;
END_REGION

REGION Network 17: Watchdog Bit Reset
   IF #Aon THEN #SEND_DATA_STAT_VAR.Watchdog := FALSE; END_IF;
END_REGION

REGION Network 18: Internal Acknowledge
   // >>>>>>>Automatic Dep_CMD when use of block interface<<<<<<
   #CMD_Acknowledge := #FP_CMD.AckAlarm;
   IF #FP_CMD.AckAlarm THEN #FP_CMD.AckAlarm := FALSE; END_IF;
END_REGION

REGION Network 19 (STL): Connection Enable Stat Bits
         A     #CPU00_CONN1_EN;
         =     #CPU00_CONN1_Enable;
         A     #CPU00_CONN1_Enable;
         O(;
         A     #CPU00_CONN2_EN;
         =     #CPU00_CONN2_Enable;
         A     #CPU00_CONN2_Enable;
         );
         O(;
         A     #CPU01_CONN1_EN;
         =     #CPU01_CONN1_Enable;
         A     #CPU01_CONN1_Enable;
         );
         O(;
         A     #CPU01_CONN2_EN;
         =     #CPU01_CONN2_Enable;
         A     #CPU01_CONN2_Enable;
         );
         =     #DummyBool;
END_REGION

REGION Network 20: CPU00 Conn1 Delay before Auto Reconect
